LIN {X 0,Y 266.568,Z 546.014,A -85,B 0,C 180,E1 -18838.226,E2 -18838.226} C_VEL
LIN {X 0,Y 268.431,Z 533.162,A -85,B 0,C 180,E1 -18839.08,E2 -18839.08} C_VEL
LIN {X 0,Y 269.683,Z 519.419,A -85,B 0,C 180,E1 -18839.681,E2 -18839.681} C_VEL
LIN {X 0,Y 272.28,Z 465.583,A -85,B 0,C 180,E1 -18841.276,E2 -18841.276} C_VEL
LIN {X 0,Y 269.856,Z 447.877,A -85,B 0,C 180,E1 -18842.351,E2 -18842.351} C_VEL
LIN {X 0,Y 266.008,Z 438.603,A -85,B 0,C 180,E1 -18843.407,E2 -18843.407} C_VEL
LIN {X 0,Y 260.297,Z 427.047,A -85,B 0,C 180,E1 -18844.98,E2 -18844.98} C_VEL
LIN {X 0,Y 255.085,Z 417.615,A -85,B 0,C 180,E1 -18846.5,E2 -18846.5} C_VEL
LIN {X 0,Y 252.805,Z 413.559,A -85,B 0,C 180,E1 -18847.202,E2 -18847.202} C_VEL
LIN {X 0,Y 252.646,Z 413.143,A -85,B 0,C 180,E1 -18847.286,E2 -18847.286} C_VEL
LIN {X 0,Y 250.833,Z 406.63,A -85,B 0,C 180,E1 -18850.843,E2 -18850.843} C_VEL
LIN {X 0,Y 249.024,Z 400.464,A -85,B 0,C 180,E1 -18854.742,E2 -18854.742} C_VEL
LIN {X 0,Y 249.022,Z 400.462,A -85,B 0,C 180,E1 -18857.364,E2 -18857.364} C_VEL
LIN {X 0,Y 249.05,Z 400.458,A -85,B 0,C 180,E1 -18862.201,E2 -18862.201} C_VEL
LIN {X 0,Y 249.05,Z 400.455,A -85,B 0,C 180,E1 -18865.64,E2 -18865.64} C_VEL
LIN {X 0,Y 249.058,Z 400.45,A -85,B 0,C 180,E1 -18869.474,E2 -18869.474} C_VEL
LIN {X 0,Y 249.08,Z 400.447,A -85,B 0,C 180,E1 -18873.163,E2 -18873.163} C_VEL
LIN {X 0,Y 249.086,Z 400.448,A -85,B 0,C 180,E1 -18876.733,E2 -18876.733} C_VEL
LIN {X 0,Y 249.118,Z 400.448,A -85,B 0,C 180,E1 -18880.212,E2 -18880.212} C_VEL
LIN {X 0,Y 249.25,Z 400.438,A -85,B 0,C 180,E1 -18883.622,E2 -18883.622} C_VEL
LIN {X 0,Y 249.26,Z 400.428,A -85,B 0,C 180,E1 -18888.617,E2 -18888.617} C_VEL
LIN {X 0,Y 249.489,Z 400.407,A -85,B 0,C 180,E1 -18891.903,E2 -18891.903} C_VEL
LIN {X 0,Y 249.442,Z 400.404,A -85,B 0,C 180,E1 -18896.77,E2 -18896.77} C_VEL
LIN {X 0,Y 249.729,Z 400.371,A -85,B 0,C 180,E1 -18900,E2 -18900} C_VEL
LIN {X 0,Y 249.442,Z 400.409,A -85,B 0,C 180,E1 -18903.23,E2 -18903.23} C_VEL
LIN {X 0,Y 249.488,Z 400.411,A -85,B 0,C 180,E1 -18908.097,E2 -18908.097} C_VEL
LIN {X 0,Y 249.273,Z 400.636,A -85,B 0,C 180,E1 -18911.795,E2 -18911.795} C_VEL
LIN {X 0,Y 250.357,Z 404.445,A -85,B 0,C 180,E1 -18914.271,E2 -18914.271} C_VEL
LIN {X 0,Y 252.764,Z 408.423,A -85,B 0,C 180,E1 -18915.03,E2 -18915.03} C_VEL
LIN {X 0,Y 254.28,Z 410.816,A -85,B 0,C 180,E1 -18915.49,E2 -18915.49} C_VEL
LIN {X 0,Y 257.244,Z 415.568,A -85,B 0,C 180,E1 -18916.36,E2 -18916.36} C_VEL
LIN {X 0,Y 261.417,Z 422.697,A -85,B 0,C 180,E1 -18917.54,E2 -18917.54} C_VEL
LIN {X 0,Y 267.546,Z 434.619,A -85,B 0,C 180,E1 -18919.194,E2 -18919.194} C_VEL
LIN {X 0,Y 272.807,Z 446.46,A -85,B 0,C 180,E1 -18920.569,E2 -18920.569} C_VEL
LIN {X 0,Y 273.096,Z 448.123,A -85,B 0,C 180,E1 -18920.679,E2 -18920.679} C_VEL
LIN {X 0,Y 269.843,Z 511.083,A -85,B 0,C 180,E1 -18922.55,E2 -18922.55} C_VEL
LIN {X 0,Y 268.607,Z 523.953,A -85,B 0,C 180,E1 -18923.2,E2 -18923.2} C_VEL
LIN {X 0,Y 266.837,Z 537.029,A -85,B 0,C 180,E1 -18924.169,E2 -18924.169} C_VEL
LIN {X 0,Y 264.669,Z 549.571,A -85,B 0,C 180,E1 -18925.463,E2 -18925.463} C_VEL
LIN {X 0,Y 262.411,Z 560.297,A -85,B 0,C 180,E1 -18926.889,E2 -18926.889} C_VEL
LIN {X 0,Y 260.125,Z 569.604,A -85,B 0,C 180,E1 -18928.424,E2 -18928.424} C_VEL
LIN {X 0,Y 257.424,Z 579.801,A -85,B 0,C 180,E1 -18930.551,E2 -18930.551} C_VEL
LIN {X 0,Y 254.954,Z 588.054,A -85,B 0,C 180,E1 -18932.711,E2 -18932.711} C_VEL
LIN {X 0,Y 252.87,Z 594.734,A -85,B 0,C 180,E1 -18934.897,E2 -18934.897} C_VEL
LIN {X 0,Y 250.791,Z 601.307,A -85,B 0,C 180,E1 -18937.658,E2 -18937.658} C_VEL
LIN {X 0,Y 249.183,Z 606.245,A -85,B 0,C 180,E1 -18940.444,E2 -18940.444} C_VEL
LIN {X 0,Y 248.195,Z 609.318,A -85,B 0,C 180,E1 -18942.812,E2 -18942.812} C_VEL
LIN {X 0,Y 247.402,Z 611.514,A -85,B 0,C 180,E1 -18945.25,E2 -18945.25} C_VEL
LIN {X 0,Y 246.873,Z 612.802,A -85,B 0,C 180,E1 -18947.746,E2 -18947.746} C_VEL
LIN {X 0,Y 246.569,Z 613.141,A -85,B 0,C 180,E1 -18950.317,E2 -18950.317} C_VEL
LIN {X 0,Y 246.519,Z 612.309,A -85,B 0,C 180,E1 -18953.222,E2 -18953.222} C_VEL
LIN {X 0,Y 246.722,Z 610.589,A -85,B 0,C 180,E1 -18955.699,E2 -18955.699} C_VEL
LIN {X 0,Y 247.211,Z 607.414,A -85,B 0,C 180,E1 -18958.526,E2 -18958.526} C_VEL
LIN {X 0,Y 247.879,Z 603.161,A -85,B 0,C 180,E1 -18961.182,E2 -18961.182} C_VEL
LIN {X 0,Y 248.794,Z 597.416,A -85,B 0,C 180,E1 -18963.877,E2 -18963.877} C_VEL
LIN {X 0,Y 250.021,Z 590.494,A -85,B 0,C 180,E1 -18966.385,E2 -18966.385} C_VEL
LIN {X 0,Y 251.436,Z 582.526,A -85,B 0,C 180,E1 -18968.691,E2 -18968.691} C_VEL
LIN {X 0,Y 253.046,Z 573.529,A -85,B 0,C 180,E1 -18970.788,E2 -18970.788} C_VEL
LIN {X 0,Y 254.837,Z 562.944,A -85,B 0,C 180,E1 -18972.746,E2 -18972.746} C_VEL
LIN {X 0,Y 256.635,Z 550.86,A -85,B 0,C 180,E1 -18974.512,E2 -18974.512} C_VEL
LIN {X 0,Y 258.123,Z 539.233,A -85,B 0,C 180,E1 -18975.813,E2 -18975.813} C_VEL
LIN {X 0,Y 259.354,Z 527.106,A -85,B 0,C 180,E1 -18976.846,E2 -18976.846} C_VEL
LIN {X 0,Y 260.376,Z 514.047,A -85,B 0,C 180,E1 -18977.632,E2 -18977.632} C_VEL
LIN {X 0,Y 261.108,Z 498.432,A -85,B 0,C 180,E1 -18978.187,E2 -18978.187} C_VEL
LIN {X 0,Y 263.221,Z 439.107,A -85,B 0,C 180,E1 -18979.921,E2 -18979.921} C_VEL
LIN {X 0,Y 259.774,Z 428.453,A -85,B 0,C 180,E1 -18980.596,E2 -18980.596} C_VEL
LIN {X 0,Y 250.616,Z 404.516,A -85,B 0,C 180,E1 -18982.343,E2 -18982.343} C_VEL
LIN {X 0,Y 249.821,Z 402.222,A -85,B 0,C 180,E1 -18982.522,E2 -18982.522} C_VEL
LIN {X 0,Y 249.445,Z 400.414,A -85,B 0,C 180,E1 -18983.324,E2 -18983.324} C_VEL
LIN {X 0,Y 249.679,Z 400.388,A -85,B 0,C 180,E1 -18988.385,E2 -18988.385} C_VEL
LIN {X 0,Y 249.68,Z 400.385,A -85,B 0,C 180,E1 -18991.611,E2 -18991.611} C_VEL
LIN {X 0,Y 249.464,Z 400.408,A -85,B 0,C 180,E1 -18996.468,E2 -18996.468} C_VEL
LIN {X 0,Y 249.426,Z 400.416,A -85,B 0,C 180,E1 -18999.731,E2 -18999.731} C_VEL
LIN {X 0,Y 249.207,Z 400.443,A -85,B 0,C 180,E1 -19004.701,E2 -19004.701} C_VEL
LIN {X 0,Y 249.139,Z 400.447,A -85,B 0,C 180,E1 -19008.075,E2 -19008.075} C_VEL
LIN {X 0,Y 249.085,Z 400.455,A -85,B 0,C 180,E1 -19011.516,E2 -19011.516} C_VEL
LIN {X 0,Y 249.129,Z 400.451,A -85,B 0,C 180,E1 -19015.48,E2 -19015.48} C_VEL
LIN {X 0,Y 249.071,Z 400.45,A -85,B 0,C 180,E1 -19018.987,E2 -19018.987} C_VEL
LIN {X 0,Y 249.033,Z 400.463,A -85,B 0,C 180,E1 -19022.423,E2 -19022.423} C_VEL
LIN {X 0,Y 249.072,Z 400.458,A -85,B 0,C 180,E1 -19026.335,E2 -19026.335} C_VEL
LIN {X 0,Y 249.1,Z 400.46,A -85,B 0,C 180,E1 -19030.05,E2 -19030.05} C_VEL
LIN {X 0,Y 258.347,Z 429.773,A -85,B 0,C 180,E1 -19031.859,E2 -19031.859} C_VEL
LIN {X 0,Y 259.41,Z 437.816,A -85,B 0,C 180,E1 -19032.236,E2 -19032.236} C_VEL
LIN {X 0,Y 256.365,Z 510.289,A -85,B 0,C 180,E1 -19034.889,E2 -19034.889} C_VEL
LIN {X 0,Y 255.661,Z 522.69,A -85,B 0,C 180,E1 -19035.617,E2 -19035.617} C_VEL
LIN {X 0,Y 254.531,Z 536.31,A -85,B 0,C 180,E1 -19036.755,E2 -19036.755} C_VEL
LIN {X 0,Y 253.393,Z 547.649,A -85,B 0,C 180,E1 -19038,E2 -19038} C_VEL
LIN {X 0,Y 252.138,Z 559.069,A -85,B 0,C 180,E1 -19039.604,E2 -19039.604} C_VEL
LIN {X 0,Y 250.863,Z 569.537,A -85,B 0,C 180,E1 -19041.428,E2 -19041.428} C_VEL
LIN {X 0,Y 249.736,Z 578.18,A -85,B 0,C 180,E1 -19043.272,E2 -19043.272} C_VEL
LIN {X 0,Y 248.787,Z 587.017,A -85,B 0,C 180,E1 -19045.599,E2 -19045.599} C_VEL
LIN {X 0,Y 247.951,Z 594.174,A -85,B 0,C 180,E1 -19047.926,E2 -19047.926} C_VEL
LIN {X 0,Y 247.385,Z 599.773,A -85,B 0,C 180,E1 -19050.187,E2 -19050.187} C_VEL
LIN {X 0,Y 246.982,Z 605.008,A -85,B 0,C 180,E1 -19052.916,E2 -19052.916} C_VEL
LIN {X 0,Y 246.573,Z 608.969,A -85,B 0,C 180,E1 -19055.789,E2 -19055.789} C_VEL
LIN {X 0,Y 246.514,Z 611.155,A -85,B 0,C 180,E1 -19058.151,E2 -19058.151} C_VEL
LIN {X 0,Y 245.924,Z 612.139,A -85,B 0,C 180,E1 -19059.499,E2 -19059.499} C_VEL
LIN {X 0,Y 243.285,Z 613.028,A -85,B 0,C 180,E1 -19061.73,E2 -19061.73} C_VEL
LIN {X 0,Y 241.181,Z 613.124,A -85,B 0,C 180,E1 -19063.556,E2 -19063.556} C_VEL
LIN {X 0,Y 240.493,Z 612.898,A -85,B 0,C 180,E1 -19064.962,E2 -19064.962} C_VEL
LIN {X 0,Y 240.551,Z 612.723,A -85,B 0,C 180,E1 -19065.434,E2 -19065.434} C_VEL
LIN {X 0,Y 241.643,Z 611.334,A -85,B 0,C 180,E1 -19068.253,E2 -19068.253} C_VEL
LIN {X 0,Y 242.589,Z 609.736,A -85,B 0,C 180,E1 -19070.051,E2 -19070.051} C_VEL
LIN {X 0,Y 244.269,Z 606.633,A -85,B 0,C 180,E1 -19072.561,E2 -19072.561} C_VEL
LIN {X 0,Y 246.742,Z 601.642,A -85,B 0,C 180,E1 -19075.463,E2 -19075.463} C_VEL
LIN {X 0,Y 249.43,Z 595.792,A -85,B 0,C 180,E1 -19077.981,E2 -19077.981} C_VEL
LIN {X 0,Y 252.714,Z 588.031,A -85,B 0,C 180,E1 -19080.542,E2 -19080.542} C_VEL
LIN {X 0,Y 256.055,Z 579.512,A -85,B 0,C 180,E1 -19082.753,E2 -19082.753} C_VEL
LIN {X 0,Y 259.357,Z 570.212,A -85,B 0,C 180,E1 -19084.663,E2 -19084.663} C_VEL
LIN {X 0,Y 262.551,Z 560.035,A -85,B 0,C 180,E1 -19086.339,E2 -19086.339} C_VEL
LIN {X 0,Y 265.555,Z 548.889,A -85,B 0,C 180,E1 -19087.795,E2 -19087.795} C_VEL
LIN {X 0,Y 268.599,Z 535.466,A -85,B 0,C 180,E1 -19089.137,E2 -19089.137} C_VEL
LIN {X 0,Y 270.877,Z 522.644,A -85,B 0,C 180,E1 -19090.082,E2 -19090.082} C_VEL
LIN {X 0,Y 272.668,Z 509.13,A -85,B 0,C 180,E1 -19090.776,E2 -19090.776} C_VEL
LIN {X 0,Y 277.82,Z 456.002,A -85,B 0,C 180,E1 -19092.755,E2 -19092.755} C_VEL
LIN {X 0,Y 275.399,Z 449.786,A -85,B 0,C 180,E1 -19093.86,E2 -19093.86} C_VEL
LIN {X 0,Y 271.486,Z 442.226,A -85,B 0,C 180,E1 -19095.629,E2 -19095.629} C_VEL
LIN {X 0,Y 267.363,Z 434.936,A -85,B 0,C 180,E1 -19097.722,E2 -19097.722} C_VEL
LIN {X 0,Y 264.428,Z 430.395,A -85,B 0,C 180,E1 -19099.372,E2 -19099.372} C_VEL
LIN {X 0,Y 261.772,Z 426.449,A -85,B 0,C 180,E1 -19101.099,E2 -19101.099} C_VEL
LIN {X 0,Y 258.771,Z 422.149,A -85,B 0,C 180,E1 -19103.407,E2 -19103.407} C_VEL
LIN {X 0,Y 255.488,Z 417.838,A -85,B 0,C 180,E1 -19106.772,E2 -19106.772} C_VEL
LIN {X 0,Y 253.639,Z 416.042,A -85,B 0,C 180,E1 -19109.631,E2 -19109.631} C_VEL
LIN {X 0,Y 252.844,Z 415.227,A -85,B 0,C 180,E1 -19111.879,E2 -19111.879} C_VEL
LIN {X 0,Y 252.7,Z 415.157,A -85,B 0,C 180,E1 -19115.181,E2 -19115.181} C_VEL
LIN {X 0,Y 253.771,Z 416.505,A -85,B 0,C 180,E1 -19118.544,E2 -19118.544} C_VEL
LIN {X 0,Y 255.625,Z 418.278,A -85,B 0,C 180,E1 -19121.205,E2 -19121.205} C_VEL
LIN {X 0,Y 258.033,Z 421.957,A -85,B 0,C 180,E1 -19123.81,E2 -19123.81} C_VEL
LIN {X 0,Y 259.615,Z 423.892,A -85,B 0,C 180,E1 -19125.133,E2 -19125.133} C_VEL
LIN {X 0,Y 261.946,Z 427.27,A -85,B 0,C 180,E1 -19126.84,E2 -19126.84} C_VEL
LIN {X 0,Y 265.527,Z 432.606,A -85,B 0,C 180,E1 -19129.073,E2 -19129.073} C_VEL
LIN {X 0,Y 268.273,Z 436.986,A -85,B 0,C 180,E1 -19130.574,E2 -19130.574} C_VEL
LIN {X 0,Y 271.957,Z 443.193,A -85,B 0,C 180,E1 -19132.381,E2 -19132.381} C_VEL
LIN {X 0,Y 274.992,Z 452.547,A -85,B 0,C 180,E1 -19134.001,E2 -19134.001} C_VEL
LIN {X 0,Y 275.778,Z 455.958,A -85,B 0,C 180,E1 -19134.463,E2 -19134.463} C_VEL
LIN {X 0,Y 276.461,Z 468.834,A -85,B 0,C 180,E1 -19135.487,E2 -19135.487} C_VEL
LIN {X 0,Y 270.924,Z 524.638,A -85,B 0,C 180,E1 -19137.657,E2 -19137.657} C_VEL
LIN {X 0,Y 268.618,Z 538.606,A -85,B 0,C 180,E1 -19138.451,E2 -19138.451} C_VEL
LIN {X 0,Y 265.527,Z 552.57,A -85,B 0,C 180,E1 -19139.591,E2 -19139.591} C_VEL
LIN {X 0,Y 262.393,Z 564.674,A -85,B 0,C 180,E1 -19140.96,E2 -19140.96} C_VEL
LIN {X 0,Y 258.685,Z 576.776,A -85,B 0,C 180,E1 -19142.715,E2 -19142.715} C_VEL
LIN {X 0,Y 255.013,Z 587.409,A -85,B 0,C 180,E1 -19144.714,E2 -19144.714} C_VEL
LIN {X 0,Y 252.05,Z 595.35,A -85,B 0,C 180,E1 -19146.591,E2 -19146.591} C_VEL
LIN {X 0,Y 249.036,Z 603.053,A -85,B 0,C 180,E1 -19148.852,E2 -19148.852} C_VEL
LIN {X 0,Y 246.865,Z 608.633,A -85,B 0,C 180,E1 -19150.892,E2 -19150.892} C_VEL
LIN {X 0,Y 244.527,Z 613.978,A -85,B 0,C 180,E1 -19153.299,E2 -19153.299} C_VEL
LIN {X 0,Y 242.666,Z 618.147,A -85,B 0,C 180,E1 -19155.751,E2 -19155.751} C_VEL
LIN {X 0,Y 241.36,Z 621.281,A -85,B 0,C 180,E1 -19158.241,E2 -19158.241} C_VEL
LIN {X 0,Y 240.717,Z 622.821,A -85,B 0,C 180,E1 -19159.913,E2 -19159.913} C_VEL
LIN {X 0,Y 239.994,Z 624.652,A -85,B 0,C 180,E1 -19163.275,E2 -19163.275} C_VEL
LIN {X 0,Y 239.838,Z 624.974,A -85,B 0,C 180,E1 -19165.076,E2 -19165.076} C_VEL
LIN {X 0,Y 239.812,Z 624.837,A -85,B 0,C 180,E1 -19166.642,E2 -19166.642} C_VEL
LIN {X 0,Y 239.913,Z 626.397,A -85,B 0,C 180,E1 -19170.002,E2 -19170.002} C_VEL
LIN {X 0,Y 239.831,Z 626.688,A -85,B 0,C 180,E1 -19171.681,E2 -19171.681} C_VEL
LIN {X 0,Y 239.791,Z 626.174,A -85,B 0,C 180,E1 -19174.794,E2 -19174.794} C_VEL
LIN {X 0,Y 239.954,Z 625.13,A -85,B 0,C 180,E1 -19176.73,E2 -19176.73} C_VEL
LIN {X 0,Y 240.672,Z 622.058,A -85,B 0,C 180,E1 -19180.093,E2 -19180.093} C_VEL
LIN {X 0,Y 241.624,Z 618.594,A -85,B 0,C 180,E1 -19182.602,E2 -19182.602} C_VEL
LIN {X 0,Y 242.992,Z 614.064,A -85,B 0,C 180,E1 -19185.09,E2 -19185.09} C_VEL
LIN {X 0,Y 245.297,Z 607.243,A -85,B 0,C 180,E1 -19187.941,E2 -19187.941} C_VEL
LIN {X 0,Y 247.616,Z 599.356,A -85,B 0,C 180,E1 -19190.507,E2 -19190.507} C_VEL
LIN {X 0,Y 250.202,Z 590.762,A -85,B 0,C 180,E1 -19192.722,E2 -19192.722} C_VEL
LIN {X 0,Y 252.924,Z 581.377,A -85,B 0,C 180,E1 -19194.635,E2 -19194.635} C_VEL
LIN {X 0,Y 255.855,Z 569.765,A -85,B 0,C 180,E1 -19196.513,E2 -19196.513} C_VEL
LIN {X 0,Y 258.453,Z 558.012,A -85,B 0,C 180,E1 -19197.976,E2 -19197.976} C_VEL
LIN {X 0,Y 260.77,Z 545.587,A -85,B 0,C 180,E1 -19199.133,E2 -19199.133} C_VEL
LIN {X 0,Y 262.745,Z 532.643,A -85,B 0,C 180,E1 -19199.993,E2 -19199.993} C_VEL
LIN {X 0,Y 264.018,Z 518.7,A -85,B 0,C 180,E1 -19200.606,E2 -19200.606} C_VEL
LIN {X 0,Y 266.594,Z 466.135,A -85,B 0,C 180,E1 -19202.206,E2 -19202.206} C_VEL
LIN {X 0,Y 264.479,Z 450.382,A -85,B 0,C 180,E1 -19203.214,E2 -19203.214} C_VEL
LIN {X 0,Y 259.935,Z 439.758,A -85,B 0,C 180,E1 -19204.521,E2 -19204.521} C_VEL
LIN {X 0,Y 253.807,Z 427.521,A -85,B 0,C 180,E1 -19206.341,E2 -19206.341} C_VEL
LIN {X 0,Y 250.372,Z 421.599,A -85,B 0,C 180,E1 -19207.396,E2 -19207.396} C_VEL
LIN {X 0,Y 247.885,Z 417.319,A -85,B 0,C 180,E1 -19208.199,E2 -19208.199} C_VEL
LIN {X 0,Y 245.301,Z 412.722,A -85,B 0,C 180,E1 -19209.154,E2 -19209.154} C_VEL
LIN {X 0,Y 243.583,Z 406.903,A -85,B 0,C 180,E1 -19212.63,E2 -19212.63} C_VEL
LIN {X 0,Y 241.937,Z 401.348,A -85,B 0,C 180,E1 -19216.369,E2 -19216.369} C_VEL
LIN {X 0,Y 241.962,Z 401.339,A -85,B 0,C 180,E1 -19220.282,E2 -19220.282} C_VEL
LIN {X 0,Y 241.995,Z 401.342,A -85,B 0,C 180,E1 -19224.49,E2 -19224.49} C_VEL
LIN {X 0,Y 241.981,Z 401.338,A -85,B 0,C 180,E1 -19228.481,E2 -19228.481} C_VEL
LIN {X 0,Y 242.015,Z 401.332,A -85,B 0,C 180,E1 -19232.314,E2 -19232.314} C_VEL
LIN {X 0,Y 242.064,Z 401.328,A -85,B 0,C 180,E1 -19236.017,E2 -19236.017} C_VEL
LIN {X 0,Y 242.045,Z 401.336,A -85,B 0,C 180,E1 -19239.609,E2 -19239.609} C_VEL
LIN {X 0,Y 242.171,Z 401.32,A -85,B 0,C 180,E1 -19243.279,E2 -19243.279} C_VEL
LIN {X 0,Y 242.194,Z 401.311,A -85,B 0,C 180,E1 -19248.28,E2 -19248.28} C_VEL
LIN {X 0,Y 242.436,Z 401.288,A -85,B 0,C 180,E1 -19251.666,E2 -19251.666} C_VEL
LIN {X 0,Y 242.268,Z 401.308,A -85,B 0,C 180,E1 -19255.007,E2 -19255.007} C_VEL
LIN {X 0,Y 242.643,Z 401.257,A -85,B 0,C 180,E1 -19258.34,E2 -19258.34} C_VEL
LIN {X 0,Y 242.643,Z 401.257,A -85,B 0,C 180,E1 -19261.66,E2 -19261.66} C_VEL
LIN {X 0,Y 242.437,Z 401.281,A -85,B 0,C 180,E1 -19266.722,E2 -19266.722} C_VEL
LIN {X 0,Y 242.34,Z 401.329,A -85,B 0,C 180,E1 -19270.021,E2 -19270.021} C_VEL
LIN {X 0,Y 243.262,Z 404.963,A -85,B 0,C 180,E1 -19272.453,E2 -19272.453} C_VEL
LIN {X 0,Y 246.064,Z 409.288,A -85,B 0,C 180,E1 -19273.419,E2 -19273.419} C_VEL
LIN {X 0,Y 250.565,Z 416.308,A -85,B 0,C 180,E1 -19274.882,E2 -19274.882} C_VEL
LIN {X 0,Y 255.602,Z 424.606,A -85,B 0,C 180,E1 -19276.401,E2 -19276.401} C_VEL
LIN {X 0,Y 261.988,Z 436.923,A -85,B 0,C 180,E1 -19278.241,E2 -19278.241} C_VEL
LIN {X 0,Y 267.348,Z 449.096,A -85,B 0,C 180,E1 -19279.733,E2 -19279.733} C_VEL
LIN {X 0,Y 266.268,Z 472.036,A -85,B 0,C 180,E1 -19280.445,E2 -19280.445} C_VEL
LIN {X 0,Y 264.106,Z 511.487,A -85,B 0,C 180,E1 -19281.656,E2 -19281.656} C_VEL
LIN {X 0,Y 262.807,Z 524.48,A -85,B 0,C 180,E1 -19282.329,E2 -19282.329} C_VEL
LIN {X 0,Y 260.98,Z 537.375,A -85,B 0,C 180,E1 -19283.305,E2 -19283.305} C_VEL
LIN {X 0,Y 258.833,Z 549.258,A -85,B 0,C 180,E1 -19284.544,E2 -19284.544} C_VEL
LIN {X 0,Y 256.412,Z 560.221,A -85,B 0,C 180,E1 -19286.011,E2 -19286.011} C_VEL
LIN {X 0,Y 253.916,Z 570.012,A -85,B 0,C 180,E1 -19287.657,E2 -19287.657} C_VEL
LIN {X 0,Y 251.461,Z 578.97,A -85,B 0,C 180,E1 -19289.55,E2 -19289.55} C_VEL
LIN {X 0,Y 248.545,Z 588.123,A -85,B 0,C 180,E1 -19291.97,E2 -19291.97} C_VEL
LIN {X 0,Y 246.355,Z 594.734,A -85,B 0,C 180,E1 -19294.173,E2 -19294.173} C_VEL
LIN {X 0,Y 244.518,Z 600.118,A -85,B 0,C 180,E1 -19296.408,E2 -19296.408} C_VEL
LIN {X 0,Y 243.058,Z 604.453,A -85,B 0,C 180,E1 -19298.672,E2 -19298.672} C_VEL
LIN {X 0,Y 241.399,Z 609.18,A -85,B 0,C 180,E1 -19302.038,E2 -19302.038} C_VEL
LIN {X 0,Y 240.507,Z 611.498,A -85,B 0,C 180,E1 -19304.533,E2 -19304.533} C_VEL
LIN {X 0,Y 239.816,Z 613.053,A -85,B 0,C 180,E1 -19307.618,E2 -19307.618} C_VEL
LIN {X 0,Y 239.507,Z 613.374,A -85,B 0,C 180,E1 -19309.79,E2 -19309.79} C_VEL
LIN {X 0,Y 239.401,Z 612.831,A -85,B 0,C 180,E1 -19312.433,E2 -19312.433} C_VEL
LIN {X 0,Y 239.572,Z 611.171,A -85,B 0,C 180,E1 -19315.226,E2 -19315.226} C_VEL
LIN {X 0,Y 240.037,Z 608.096,A -85,B 0,C 180,E1 -19318.193,E2 -19318.193} C_VEL
LIN {X 0,Y 240.751,Z 603.639,A -85,B 0,C 180,E1 -19321.136,E2 -19321.136} C_VEL
LIN {X 0,Y 241.6,Z 598.536,A -85,B 0,C 180,E1 -19323.663,E2 -19323.663} C_VEL
LIN {X 0,Y 242.722,Z 592.355,A -85,B 0,C 180,E1 -19326.084,E2 -19326.084} C_VEL
LIN {X 0,Y 244.122,Z 584.751,A -85,B 0,C 180,E1 -19328.464,E2 -19328.464} C_VEL
LIN {X 0,Y 245.781,Z 575.944,A -85,B 0,C 180,E1 -19330.67,E2 -19330.67} C_VEL
LIN {X 0,Y 247.518,Z 566.141,A -85,B 0,C 180,E1 -19332.652,E2 -19332.652} C_VEL
LIN {X 0,Y 249.188,Z 555.878,A -85,B 0,C 180,E1 -19334.32,E2 -19334.32} C_VEL
LIN {X 0,Y 250.807,Z 544.253,A -85,B 0,C 180,E1 -19335.805,E2 -19335.805} C_VEL
LIN {X 0,Y 252.27,Z 531.643,A -85,B 0,C 180,E1 -19337.037,E2 -19337.037} C_VEL
LIN {X 0,Y 253.431,Z 518.677,A -85,B 0,C 180,E1 -19337.943,E2 -19337.943} C_VEL
LIN {X 0,Y 254.242,Z 505.414,A -85,B 0,C 180,E1 -19338.538,E2 -19338.538} C_VEL
LIN {X 0,Y 256.641,Z 440.017,A -85,B 0,C 180,E1 -19340.51,E2 -19340.51} C_VEL
LIN {X 0,Y 248.497,Z 417.323,A -85,B 0,C 180,E1 -19342.116,E2 -19342.116} C_VEL
LIN {X 0,Y 242.596,Z 402.349,A -85,B 0,C 180,E1 -19343.344,E2 -19343.344} C_VEL
LIN {X 0,Y 242.359,Z 401.297,A -85,B 0,C 180,E1 -19343.859,E2 -19343.859} C_VEL
LIN {X 0,Y 242.639,Z 401.265,A -85,B 0,C 180,E1 -19348.338,E2 -19348.338} C_VEL
LIN {X 0,Y 242.64,Z 401.262,A -85,B 0,C 180,E1 -19351.658,E2 -19351.658} C_VEL
LIN {X 0,Y 242.437,Z 401.282,A -85,B 0,C 180,E1 -19356.657,E2 -19356.657} C_VEL
LIN {X 0,Y 242.347,Z 401.3,A -85,B 0,C 180,E1 -19360.018,E2 -19360.018} C_VEL
LIN {X 0,Y 242.168,Z 401.319,A -85,B 0,C 180,E1 -19365.138,E2 -19365.138} C_VEL
LIN {X 0,Y 242.072,Z 401.323,A -85,B 0,C 180,E1 -19368.622,E2 -19368.622} C_VEL
LIN {X 0,Y 242.011,Z 401.34,A -85,B 0,C 180,E1 -19372.178,E2 -19372.178} C_VEL
LIN {X 0,Y 242.065,Z 401.326,A -85,B 0,C 180,E1 -19375.836,E2 -19375.836} C_VEL
LIN {X 0,Y 242.005,Z 401.333,A -85,B 0,C 180,E1 -19379.581,E2 -19379.581} C_VEL
LIN {X 0,Y 241.988,Z 401.343,A -85,B 0,C 180,E1 -19383.488,E2 -19383.488} C_VEL
LIN {X 0,Y 242.01,Z 401.341,A -85,B 0,C 180,E1 -19387.575,E2 -19387.575} C_VEL
LIN {X 0,Y 242.044,Z 401.339,A -85,B 0,C 180,E1 -19389.545,E2 -19389.545} C_VEL
LIN {X 0,Y 249.887,Z 425.715,A -85,B 0,C 180,E1 -19391.133,E2 -19391.133} C_VEL
LIN {X 0,Y 251.825,Z 432.71,A -85,B 0,C 180,E1 -19391.546,E2 -19391.546} C_VEL
LIN {X 0,Y 252.582,Z 438.328,A -85,B 0,C 180,E1 -19391.818,E2 -19391.818} C_VEL
LIN {X 0,Y 249.442,Z 510.774,A -85,B 0,C 180,E1 -19394.56,E2 -19394.56} C_VEL
LIN {X 0,Y 248.664,Z 523.331,A -85,B 0,C 180,E1 -19395.328,E2 -19395.328} C_VEL
LIN {X 0,Y 247.528,Z 536.734,A -85,B 0,C 180,E1 -19396.486,E2 -19396.486} C_VEL
LIN {X 0,Y 246.27,Z 548.996,A -85,B 0,C 180,E1 -19397.897,E2 -19397.897} C_VEL
LIN {X 0,Y 245.003,Z 560.145,A -85,B 0,C 180,E1 -19399.533,E2 -19399.533} C_VEL
LIN {X 0,Y 243.749,Z 570.254,A -85,B 0,C 180,E1 -19401.369,E2 -19401.369} C_VEL
LIN {X 0,Y 242.489,Z 579.841,A -85,B 0,C 180,E1 -19403.537,E2 -19403.537} C_VEL
LIN {X 0,Y 241.527,Z 588.431,A -85,B 0,C 180,E1 -19405.934,E2 -19405.934} C_VEL
LIN {X 0,Y 240.719,Z 595.238,A -85,B 0,C 180,E1 -19408.296,E2 -19408.296} C_VEL
LIN {X 0,Y 240.208,Z 601.145,A -85,B 0,C 180,E1 -19410.875,E2 -19410.875} C_VEL
LIN {X 0,Y 239.713,Z 606.438,A -85,B 0,C 180,E1 -19413.91,E2 -19413.91} C_VEL
LIN {X 0,Y 239.504,Z 608.808,A -85,B 0,C 180,E1 -19415.744,E2 -19415.744} C_VEL
LIN {X 0,Y 239.398,Z 611.078,A -85,B 0,C 180,E1 -19418.16,E2 -19418.16} C_VEL
LIN {X 0,Y 239.51,Z 612.221,A -85,B 0,C 180,E1 -19419.874,E2 -19419.874} C_VEL
LIN {X 0,Y 239.946,Z 613.112,A -85,B 0,C 180,E1 -19422.968,E2 -19422.968} C_VEL
LIN {X 0,Y 240.551,Z 612.723,A -85,B 0,C 180,E1 -19425.434,E2 -19425.434} C_VEL
LIN {X 0,Y 240.37,Z 612.261,A -85,B 0,C 180,E1 -19426.836,E2 -19426.836} C_VEL
LIN {X 0,Y 238.52,Z 611.009,A -85,B 0,C 180,E1 -19429.152,E2 -19429.152} C_VEL
LIN {X 0,Y 237.004,Z 609.191,A -85,B 0,C 180,E1 -19431.472,E2 -19431.472} C_VEL
LIN {X 0,Y 237.339,Z 607.608,A -85,B 0,C 180,E1 -19432.846,E2 -19432.846} C_VEL
LIN {X 0,Y 239.666,Z 603.432,A -85,B 0,C 180,E1 -19435.541,E2 -19435.541} C_VEL
LIN {X 0,Y 242.621,Z 597.494,A -85,B 0,C 180,E1 -19438.34,E2 -19438.34} C_VEL
LIN {X 0,Y 246,Z 590.388,A -85,B 0,C 180,E1 -19440.911,E2 -19440.911} C_VEL
LIN {X 0,Y 249.504,Z 582.136,A -85,B 0,C 180,E1 -19443.229,E2 -19443.229} C_VEL
LIN {X 0,Y 253.385,Z 572.109,A -85,B 0,C 180,E1 -19445.431,E2 -19445.431} C_VEL
LIN {X 0,Y 257.008,Z 561.408,A -85,B 0,C 180,E1 -19447.266,E2 -19447.266} C_VEL
LIN {X 0,Y 260.176,Z 550.665,A -85,B 0,C 180,E1 -19448.74,E2 -19448.74} C_VEL
LIN {X 0,Y 263.144,Z 538.765,A -85,B 0,C 180,E1 -19449.998,E2 -19449.998} C_VEL
LIN {X 0,Y 265.826,Z 525.23,A -85,B 0,C 180,E1 -19451.077,E2 -19451.077} C_VEL
LIN {X 0,Y 267.802,Z 511.666,A -85,B 0,C 180,E1 -19451.819,E2 -19451.819} C_VEL
LIN {X 0,Y 273.357,Z 458.874,A -85,B 0,C 180,E1 -19453.832,E2 -19453.832} C_VEL
LIN {X 0,Y 270.772,Z 452.622,A -85,B 0,C 180,E1 -19455.072,E2 -19455.072} C_VEL
LIN {X 0,Y 266.891,Z 445.109,A -85,B 0,C 180,E1 -19457.019,E2 -19457.019} C_VEL
LIN {X 0,Y 263.865,Z 439.602,A -85,B 0,C 180,E1 -19458.744,E2 -19458.744} C_VEL
LIN {X 0,Y 261.787,Z 436.366,A -85,B 0,C 180,E1 -19460.02,E2 -19460.02} C_VEL
LIN {X 0,Y 259.543,Z 432.863,A -85,B 0,C 180,E1 -19461.555,E2 -19461.555} C_VEL
LIN {X 0,Y 256.667,Z 428.644,A -85,B 0,C 180,E1 -19463.901,E2 -19463.901} C_VEL
LIN {X 0,Y 253.731,Z 424.52,A -85,B 0,C 180,E1 -19467.195,E2 -19467.195} C_VEL
LIN {X 0,Y 251.982,Z 422.789,A -85,B 0,C 180,E1 -19470.166,E2 -19470.166} C_VEL
LIN {X 0,Y 251.252,Z 422.055,A -85,B 0,C 180,E1 -19472.953,E2 -19472.953} C_VEL
LIN {X 0,Y 251.404,Z 422.303,A -85,B 0,C 180,E1 -19475.948,E2 -19475.948} C_VEL
LIN {X 0,Y 253.539,Z 424.567,A -85,B 0,C 180,E1 -19480.376,E2 -19480.376} C_VEL
LIN {X 0,Y 254.089,Z 425.443,A -85,B 0,C 180,E1 -19481.147,E2 -19481.147} C_VEL
LIN {X 0,Y 256.599,Z 429.109,A -85,B 0,C 180,E1 -19483.852,E2 -19483.852} C_VEL
LIN {X 0,Y 257.638,Z 430.512,A -85,B 0,C 180,E1 -19484.752,E2 -19484.752} C_VEL
LIN {X 0,Y 260.994,Z 435.664,A -85,B 0,C 180,E1 -19487.281,E2 -19487.281} C_VEL
LIN {X 0,Y 263.165,Z 439.105,A -85,B 0,C 180,E1 -19488.662,E2 -19488.662} C_VEL
LIN {X 0,Y 265.862,Z 443.65,A -85,B 0,C 180,E1 -19490.227,E2 -19490.227} C_VEL
LIN {X 0,Y 268.745,Z 448.915,A -85,B 0,C 180,E1 -19491.73,E2 -19491.73} C_VEL
LIN {X 0,Y 271.591,Z 458.563,A -85,B 0,C 180,E1 -19493.394,E2 -19493.394} C_VEL
LIN {X 0,Y 272.014,Z 470.266,A -85,B 0,C 180,E1 -19494.36,E2 -19494.36} C_VEL
LIN {X 0,Y 266.398,Z 523.966,A -85,B 0,C 180,E1 -19496.473,E2 -19496.473} C_VEL
LIN {X 0,Y 264.004,Z 537.881,A -85,B 0,C 180,E1 -19497.269,E2 -19497.269} C_VEL
LIN {X 0,Y 260.976,Z 550.939,A -85,B 0,C 180,E1 -19498.326,E2 -19498.326} C_VEL
LIN {X 0,Y 257.631,Z 563.395,A -85,B 0,C 180,E1 -19499.693,E2 -19499.693} C_VEL
LIN {X 0,Y 253.677,Z 575.657,A -85,B 0,C 180,E1 -19501.454,E2 -19501.454} C_VEL
LIN {X 0,Y 250.105,Z 585.524,A -85,B 0,C 180,E1 -19503.284,E2 -19503.284} C_VEL
LIN {X 0,Y 246.251,Z 595.175,A -85,B 0,C 180,E1 -19505.557,E2 -19505.557} C_VEL
LIN {X 0,Y 242.914,Z 603.046,A -85,B 0,C 180,E1 -19507.909,E2 -19507.909} C_VEL
LIN {X 0,Y 240.216,Z 609.367,A -85,B 0,C 180,E1 -19510.341,E2 -19510.341} C_VEL
LIN {X 0,Y 237.769,Z 614.48,A -85,B 0,C 180,E1 -19512.81,E2 -19512.81} C_VEL
LIN {X 0,Y 235.773,Z 618.484,A -85,B 0,C 180,E1 -19515.325,E2 -19515.325} C_VEL
LIN {X 0,Y 234.393,Z 621.451,A -85,B 0,C 180,E1 -19517.887,E2 -19517.887} C_VEL
LIN {X 0,Y 233.219,Z 623.918,A -85,B 0,C 180,E1 -19521.336,E2 -19521.336} C_VEL
LIN {X 0,Y 232.921,Z 624.555,A -85,B 0,C 180,E1 -19523.07,E2 -19523.07} C_VEL
LIN {X 0,Y 232.731,Z 624.722,A -85,B 0,C 180,E1 -19525.228,E2 -19525.228} C_VEL
LIN {X 0,Y 232.731,Z 624.569,A -85,B 0,C 180,E1 -19526.973,E2 -19526.973} C_VEL
LIN {X 0,Y 232.822,Z 626.146,A -85,B 0,C 180,E1 -19530.002,E2 -19530.002} C_VEL
LIN {X 0,Y 232.742,Z 626.469,A -85,B 0,C 180,E1 -19531.733,E2 -19531.733} C_VEL
LIN {X 0,Y 232.732,Z 625.938,A -85,B 0,C 180,E1 -19535.2,E2 -19535.2} C_VEL
LIN {X 0,Y 232.892,Z 625.043,A -85,B 0,C 180,E1 -19536.935,E2 -19536.935} C_VEL
LIN {X 0,Y 233.67,Z 622.038,A -85,B 0,C 180,E1 -19540.399,E2 -19540.399} C_VEL
LIN {X 0,Y 234.66,Z 618.643,A -85,B 0,C 180,E1 -19542.983,E2 -19542.983} C_VEL
LIN {X 0,Y 236.151,Z 614.186,A -85,B 0,C 180,E1 -19545.538,E2 -19545.538} C_VEL
LIN {X 0,Y 238.553,Z 607.516,A -85,B 0,C 180,E1 -19548.466,E2 -19548.466} C_VEL
LIN {X 0,Y 240.901,Z 600.076,A -85,B 0,C 180,E1 -19551.003,E2 -19551.003} C_VEL
LIN {X 0,Y 243.695,Z 591.296,A -85,B 0,C 180,E1 -19553.364,E2 -19553.364} C_VEL
LIN {X 0,Y 246.54,Z 582.116,A -85,B 0,C 180,E1 -19555.317,E2 -19555.317} C_VEL
LIN {X 0,Y 249.578,Z 570.707,A -85,B 0,C 180,E1 -19557.234,E2 -19557.234} C_VEL
LIN {X 0,Y 252.275,Z 559.283,A -85,B 0,C 180,E1 -19558.724,E2 -19558.724} C_VEL
LIN {X 0,Y 254.848,Z 546.283,A -85,B 0,C 180,E1 -19559.991,E2 -19559.991} C_VEL
LIN {X 0,Y 256.875,Z 533.72,A -85,B 0,C 180,E1 -19560.865,E2 -19560.865} C_VEL
LIN {X 0,Y 258.292,Z 520.295,A -85,B 0,C 180,E1 -19561.502,E2 -19561.502} C_VEL
LIN {X 0,Y 261.135,Z 467.707,A -85,B 0,C 180,E1 -19563.133,E2 -19563.133} C_VEL
LIN {X 0,Y 259.301,Z 453.36,A -85,B 0,C 180,E1 -19564.075,E2 -19564.075} C_VEL
LIN {X 0,Y 255.078,Z 443.476,A -85,B 0,C 180,E1 -19565.354,E2 -19565.354} C_VEL
LIN {X 0,Y 249.295,Z 431.757,A -85,B 0,C 180,E1 -19567.175,E2 -19567.175} C_VEL
LIN {X 0,Y 244.323,Z 422.817,A -85,B 0,C 180,E1 -19568.837,E2 -19568.837} C_VEL
LIN {X 0,Y 241.013,Z 417.544,A -85,B 0,C 180,E1 -19569.992,E2 -19569.992} C_VEL
LIN {X 0,Y 238.266,Z 413.211,A -85,B 0,C 180,E1 -19571.007,E2 -19571.007} C_VEL
LIN {X 0,Y 237.888,Z 412.305,A -85,B 0,C 180,E1 -19571.278,E2 -19571.278} C_VEL
LIN {X 0,Y 236.489,Z 407.369,A -85,B 0,C 180,E1 -19574.501,E2 -19574.501} C_VEL
LIN {X 0,Y 234.889,Z 402.228,A -85,B 0,C 180,E1 -19578.421,E2 -19578.421} C_VEL
LIN {X 0,Y 234.925,Z 402.221,A -85,B 0,C 180,E1 -19581.08,E2 -19581.08} C_VEL
LIN {X 0,Y 234.937,Z 402.214,A -85,B 0,C 180,E1 -19585.363,E2 -19585.363} C_VEL
LIN {X 0,Y 234.938,Z 402.209,A -85,B 0,C 180,E1 -19589.433,E2 -19589.433} C_VEL
LIN {X 0,Y 235.001,Z 402.201,A -85,B 0,C 180,E1 -19593.795,E2 -19593.795} C_VEL
LIN {X 0,Y 235.019,Z 402.209,A -85,B 0,C 180,E1 -19598.971,E2 -19598.971} C_VEL
LIN {X 0,Y 235.104,Z 402.199,A -85,B 0,C 180,E1 -19603.06,E2 -19603.06} C_VEL
LIN {X 0,Y 235.154,Z 402.191,A -85,B 0,C 180,E1 -19607.924,E2 -19607.924} C_VEL
LIN {X 0,Y 235.385,Z 402.165,A -85,B 0,C 180,E1 -19611.414,E2 -19611.414} C_VEL
LIN {X 0,Y 235.412,Z 402.15,A -85,B 0,C 180,E1 -19613.142,E2 -19613.142} C_VEL
LIN {X 0,Y 235.603,Z 402.133,A -85,B 0,C 180,E1 -19618.291,E2 -19618.291} C_VEL
LIN {X 0,Y 235.603,Z 402.134,A -85,B 0,C 180,E1 -19621.71,E2 -19621.71} C_VEL
LIN {X 0,Y 235.384,Z 402.166,A -85,B 0,C 180,E1 -19627.938,E2 -19627.938} C_VEL
LIN {X 0,Y 236.155,Z 405.311,A -85,B 0,C 180,E1 -19630.394,E2 -19630.394} C_VEL
LIN {X 0,Y 238.23,Z 408.723,A -85,B 0,C 180,E1 -19631.217,E2 -19631.217} C_VEL
LIN {X 0,Y 240.051,Z 411.067,A -85,B 0,C 180,E1 -19631.88,E2 -19631.88} C_VEL
LIN {X 0,Y 246.088,Z 420.27,A -85,B 0,C 180,E1 -19633.97,E2 -19633.97} C_VEL
LIN {X 0,Y 252.467,Z 431.309,A -85,B 0,C 180,E1 -19636.008,E2 -19636.008} C_VEL
LIN {X 0,Y 258.155,Z 442.889,A -85,B 0,C 180,E1 -19637.739,E2 -19637.739} C_VEL
LIN {X 0,Y 261.952,Z 451.736,A -85,B 0,C 180,E1 -19638.844,E2 -19638.844} C_VEL
LIN {X 0,Y 258.526,Z 511.52,A -85,B 0,C 180,E1 -19640.696,E2 -19640.696} C_VEL
LIN {X 0,Y 257.175,Z 524.358,A -85,B 0,C 180,E1 -19641.367,E2 -19641.367} C_VEL
LIN {X 0,Y 255.276,Z 537.214,A -85,B 0,C 180,E1 -19642.347,E2 -19642.347} C_VEL
LIN {X 0,Y 253.066,Z 548.954,A -85,B 0,C 180,E1 -19643.583,E2 -19643.583} C_VEL
LIN {X 0,Y 250.541,Z 559.903,A -85,B 0,C 180,E1 -19645.056,E2 -19645.056} C_VEL
LIN {X 0,Y 247.834,Z 570.187,A -85,B 0,C 180,E1 -19646.809,E2 -19646.809} C_VEL
LIN {X 0,Y 245.35,Z 578.678,A -85,B 0,C 180,E1 -19648.616,E2 -19648.616} C_VEL
LIN {X 0,Y 242.544,Z 587.171,A -85,B 0,C 180,E1 -19650.859,E2 -19650.859} C_VEL
LIN {X 0,Y 240.092,Z 594.064,A -85,B 0,C 180,E1 -19653.134,E2 -19653.134} C_VEL
LIN {X 0,Y 238.072,Z 599.712,A -85,B 0,C 180,E1 -19655.475,E2 -19655.475} C_VEL
LIN {X 0,Y 236.445,Z 604.262,A -85,B 0,C 180,E1 -19657.857,E2 -19657.857} C_VEL
LIN {X 0,Y 235.098,Z 607.838,A -85,B 0,C 180,E1 -19660.254,E2 -19660.254} C_VEL
LIN {X 0,Y 234.04,Z 610.481,A -85,B 0,C 180,E1 -19662.63,E2 -19662.63} C_VEL
LIN {X 0,Y 233.001,Z 612.811,A -85,B 0,C 180,E1 -19666.07,E2 -19666.07} C_VEL
LIN {X 0,Y 232.472,Z 613.554,A -85,B 0,C 180,E1 -19669.095,E2 -19669.095} C_VEL
LIN {X 0,Y 232.301,Z 613.158,A -85,B 0,C 180,E1 -19671.869,E2 -19671.869} C_VEL
LIN {X 0,Y 232.436,Z 611.528,A -85,B 0,C 180,E1 -19674.934,E2 -19674.934} C_VEL
LIN {X 0,Y 232.825,Z 608.924,A -85,B 0,C 180,E1 -19677.694,E2 -19677.694} C_VEL
LIN {X 0,Y 233.38,Z 605.784,A -85,B 0,C 180,E1 -19680.041,E2 -19680.041} C_VEL
LIN {X 0,Y 234.353,Z 599.98,A -85,B 0,C 180,E1 -19683.265,E2 -19683.265} C_VEL
LIN {X 0,Y 235.695,Z 592.751,A -85,B 0,C 180,E1 -19686.26,E2 -19686.26} C_VEL
LIN {X 0,Y 237.122,Z 585.214,A -85,B 0,C 180,E1 -19688.709,E2 -19688.709} C_VEL
LIN {X 0,Y 238.944,Z 575.839,A -85,B 0,C 180,E1 -19691.121,E2 -19691.121} C_VEL
LIN {X 0,Y 240.869,Z 565.406,A -85,B 0,C 180,E1 -19693.262,E2 -19693.262} C_VEL
LIN {X 0,Y 242.715,Z 553.922,A -85,B 0,C 180,E1 -19695.107,E2 -19695.107} C_VEL
LIN {X 0,Y 244.425,Z 542.051,A -85,B 0,C 180,E1 -19696.594,E2 -19696.594} C_VEL
LIN {X 0,Y 245.815,Z 529.628,A -85,B 0,C 180,E1 -19697.769,E2 -19697.769} C_VEL
LIN {X 0,Y 246.994,Z 516.182,A -85,B 0,C 180,E1 -19698.665,E2 -19698.665} C_VEL
LIN {X 0,Y 247.746,Z 502.926,A -85,B 0,C 180,E1 -19699.217,E2 -19699.217} C_VEL
LIN {X 0,Y 250.092,Z 441.448,A -85,B 0,C 180,E1 -19701.112,E2 -19701.112} C_VEL
LIN {X 0,Y 240.933,Z 416.334,A -85,B 0,C 180,E1 -19702.966,E2 -19702.966} C_VEL
LIN {X 0,Y 235.968,Z 404.432,A -85,B 0,C 180,E1 -19703.98,E2 -19703.98} C_VEL
LIN {X 0,Y 235.346,Z 402.6,A -85,B 0,C 180,E1 -19704.16,E2 -19704.16} C_VEL
LIN {X 0,Y 235.246,Z 402.181,A -85,B 0,C 180,E1 -19704.426,E2 -19704.426} C_VEL
LIN {X 0,Y 235.598,Z 402.142,A -85,B 0,C 180,E1 -19708.288,E2 -19708.288} C_VEL
LIN {X 0,Y 235.6,Z 402.14,A -85,B 0,C 180,E1 -19711.707,E2 -19711.707} C_VEL
LIN {X 0,Y 235.408,Z 402.157,A -85,B 0,C 180,E1 -19716.856,E2 -19716.856} C_VEL
LIN {X 0,Y 235.255,Z 402.182,A -85,B 0,C 180,E1 -19720.323,E2 -19720.323} C_VEL
LIN {X 0,Y 235.114,Z 402.199,A -85,B 0,C 180,E1 -19725.604,E2 -19725.604} C_VEL
LIN {X 0,Y 235.008,Z 402.203,A -85,B 0,C 180,E1 -19729.203,E2 -19729.203} C_VEL
LIN {X 0,Y 234.959,Z 402.216,A -85,B 0,C 180,E1 -19732.88,E2 -19732.88} C_VEL
LIN {X 0,Y 234.966,Z 402.206,A -85,B 0,C 180,E1 -19736.655,E2 -19736.655} C_VEL
LIN {X 0,Y 234.92,Z 402.218,A -85,B 0,C 180,E1 -19740.566,E2 -19740.566} C_VEL
LIN {X 0,Y 234.957,Z 402.216,A -85,B 0,C 180,E1 -19744.63,E2 -19744.63} C_VEL
LIN {X 0,Y 234.999,Z 402.212,A -85,B 0,C 180,E1 -19749.026,E2 -19749.026} C_VEL
LIN {X 0,Y 240.929,Z 420.062,A -85,B 0,C 180,E1 -19750.261,E2 -19750.261} C_VEL
LIN {X 0,Y 245.072,Z 433.85,A -85,B 0,C 180,E1 -19751.128,E2 -19751.128} C_VEL
LIN {X 0,Y 245.736,Z 439.338,A -85,B 0,C 180,E1 -19751.401,E2 -19751.401} C_VEL
LIN {X 0,Y 242.539,Z 510.325,A -85,B 0,C 180,E1 -19754.178,E2 -19754.178} C_VEL
LIN {X 0,Y 241.697,Z 523.629,A -85,B 0,C 180,E1 -19755.012,E2 -19755.012} C_VEL
LIN {X 0,Y 240.52,Z 537.185,A -85,B 0,C 180,E1 -19756.227,E2 -19756.227} C_VEL
LIN {X 0,Y 239.349,Z 548.187,A -85,B 0,C 180,E1 -19757.518,E2 -19757.518} C_VEL
LIN {X 0,Y 238.049,Z 559.561,A -85,B 0,C 180,E1 -19759.216,E2 -19759.216} C_VEL
LIN {X 0,Y 236.782,Z 569.444,A -85,B 0,C 180,E1 -19761.036,E2 -19761.036} C_VEL
LIN {X 0,Y 235.674,Z 577.592,A -85,B 0,C 180,E1 -19762.852,E2 -19762.852} C_VEL
LIN {X 0,Y 234.648,Z 586.623,A -85,B 0,C 180,E1 -19765.314,E2 -19765.314} C_VEL
LIN {X 0,Y 233.797,Z 593.828,A -85,B 0,C 180,E1 -19767.753,E2 -19767.753} C_VEL
LIN {X 0,Y 233.22,Z 599.585,A -85,B 0,C 180,E1 -19770.162,E2 -19770.162} C_VEL
LIN {X 0,Y 232.774,Z 605.025,A -85,B 0,C 180,E1 -19773.071,E2 -19773.071} C_VEL
LIN {X 0,Y 232.457,Z 607.889,A -85,B 0,C 180,E1 -19775.089,E2 -19775.089} C_VEL
LIN {X 0,Y 232.322,Z 609.887,A -85,B 0,C 180,E1 -19776.842,E2 -19776.842} C_VEL
LIN {X 0,Y 232.404,Z 612.077,A -85,B 0,C 180,E1 -19779.62,E2 -19779.62} C_VEL
LIN {X 0,Y 232.756,Z 613.182,A -85,B 0,C 180,E1 -19782.425,E2 -19782.425} C_VEL
LIN {X 0,Y 233.493,Z 613.1,A -85,B 0,C 180,E1 -19785.576,E2 -19785.576} C_VEL
LIN {X 0,Y 234.368,Z 612.218,A -85,B 0,C 180,E1 -19787.883,E2 -19787.883} C_VEL
LIN {X 0,Y 235.461,Z 610.682,A -85,B 0,C 180,E1 -19790.04,E2 -19790.04} C_VEL
LIN {X 0,Y 237.339,Z 607.608,A -85,B 0,C 180,E1 -19792.846,E2 -19792.846} C_VEL
LIN {X 0,Y 237.785,Z 605.853,A -85,B 0,C 180,E1 -19794.204,E2 -19794.204} C_VEL
LIN {X 0,Y 236.966,Z 602.77,A -85,B 0,C 180,E1 -19796.474,E2 -19796.474} C_VEL
LIN {X 0,Y 236.474,Z 599.074,A -85,B 0,C 180,E1 -19798.692,E2 -19798.692} C_VEL
LIN {X 0,Y 237.398,Z 596.343,A -85,B 0,C 180,E1 -19799.935,E2 -19799.935} C_VEL
LIN {X 0,Y 241.012,Z 588.938,A -85,B 0,C 180,E1 -19802.507,E2 -19802.507} C_VEL
LIN {X 0,Y 245.082,Z 579.928,A -85,B 0,C 180,E1 -19804.935,E2 -19804.935} C_VEL
LIN {X 0,Y 249.172,Z 569.651,A -85,B 0,C 180,E1 -19807.088,E2 -19807.088} C_VEL
LIN {X 0,Y 252.8,Z 559.289,A -85,B 0,C 180,E1 -19808.795,E2 -19808.795} C_VEL
LIN {X 0,Y 256.402,Z 547.151,A -85,B 0,C 180,E1 -19810.343,E2 -19810.343} C_VEL
LIN {X 0,Y 259.426,Z 534.964,A -85,B 0,C 180,E1 -19811.543,E2 -19811.543} C_VEL
LIN {X 0,Y 261.608,Z 523.938,A -85,B 0,C 180,E1 -19812.37,E2 -19812.37} C_VEL
LIN {X 0,Y 263.546,Z 511.246,A -85,B 0,C 180,E1 -19813.052,E2 -19813.052} C_VEL
LIN {X 0,Y 268.992,Z 461.617,A -85,B 0,C 180,E1 -19814.978,E2 -19814.978} C_VEL
LIN {X 0,Y 265.902,Z 454.616,A -85,B 0,C 180,E1 -19816.6,E2 -19816.6} C_VEL
LIN {X 0,Y 261.669,Z 446.405,A -85,B 0,C 180,E1 -19819.045,E2 -19819.045} C_VEL
LIN {X 0,Y 259.476,Z 442.728,A -85,B 0,C 180,E1 -19820.485,E2 -19820.485} C_VEL
LIN {X 0,Y 257.358,Z 439.28,A -85,B 0,C 180,E1 -19822.036,E2 -19822.036} C_VEL
LIN {X 0,Y 254.883,Z 435.395,A -85,B 0,C 180,E1 -19824.189,E2 -19824.189} C_VEL
LIN {X 0,Y 252.044,Z 431.283,A -85,B 0,C 180,E1 -19827.542,E2 -19827.542} C_VEL
LIN {X 0,Y 250.631,Z 429.826,A -85,B 0,C 180,E1 -19830.023,E2 -19830.023} C_VEL
LIN {X 0,Y 249.921,Z 429.074,A -85,B 0,C 180,E1 -19832.48,E2 -19832.48} C_VEL
LIN {X 0,Y 249.918,Z 429.125,A -85,B 0,C 180,E1 -19835.366,E2 -19835.366} C_VEL
LIN {X 0,Y 251.045,Z 430.571,A -85,B 0,C 180,E1 -19838.733,E2 -19838.733} C_VEL
LIN {X 0,Y 252.25,Z 431.904,A -85,B 0,C 180,E1 -19840.625,E2 -19840.625} C_VEL
LIN {X 0,Y 254.57,Z 435.606,A -85,B 0,C 180,E1 -19843.379,E2 -19843.379} C_VEL
LIN {X 0,Y 255.678,Z 437.226,A -85,B 0,C 180,E1 -19844.387,E2 -19844.387} C_VEL
LIN {X 0,Y 258.612,Z 441.839,A -85,B 0,C 180,E1 -19846.728,E2 -19846.728} C_VEL
LIN {X 0,Y 260.741,Z 445.518,A -85,B 0,C 180,E1 -19848.204,E2 -19848.204} C_VEL
LIN {X 0,Y 263.048,Z 449.557,A -85,B 0,C 180,E1 -19849.613,E2 -19849.613} C_VEL
LIN {X 0,Y 265.426,Z 454.046,A -85,B 0,C 180,E1 -19850.947,E2 -19850.947} C_VEL
LIN {X 0,Y 267.537,Z 461.929,A -85,B 0,C 180,E1 -19852.353,E2 -19852.353} C_VEL
LIN {X 0,Y 267.845,Z 471.546,A -85,B 0,C 180,E1 -19853.175,E2 -19853.175} C_VEL
LIN {X 0,Y 261.99,Z 523.567,A -85,B 0,C 180,E1 -19855.25,E2 -19855.25} C_VEL
LIN {X 0,Y 259.509,Z 537.444,A -85,B 0,C 180,E1 -19856.046,E2 -19856.046} C_VEL
LIN {X 0,Y 256.586,Z 549.68,A -85,B 0,C 180,E1 -19857.02,E2 -19857.02} C_VEL
LIN {X 0,Y 253.449,Z 560.843,A -85,B 0,C 180,E1 -19858.209,E2 -19858.209} C_VEL
LIN {X 0,Y 249.656,Z 572.375,A -85,B 0,C 180,E1 -19859.791,E2 -19859.791} C_VEL
LIN {X 0,Y 245.375,Z 583.704,A -85,B 0,C 180,E1 -19861.8,E2 -19861.8} C_VEL
LIN {X 0,Y 241.854,Z 592.164,A -85,B 0,C 180,E1 -19863.698,E2 -19863.698} C_VEL
LIN {X 0,Y 238.025,Z 600.725,A -85,B 0,C 180,E1 -19866.154,E2 -19866.154} C_VEL
LIN {X 0,Y 234.447,Z 608.249,A -85,B 0,C 180,E1 -19868.919,E2 -19868.919} C_VEL
LIN {X 0,Y 231.873,Z 613.535,A -85,B 0,C 180,E1 -19871.445,E2 -19871.445} C_VEL
LIN {X 0,Y 229.5,Z 617.69,A -85,B 0,C 180,E1 -19874.004,E2 -19874.004} C_VEL
LIN {X 0,Y 228.357,Z 619.859,A -85,B 0,C 180,E1 -19875.749,E2 -19875.749} C_VEL
LIN {X 0,Y 226.721,Z 622.961,A -85,B 0,C 180,E1 -19879.284,E2 -19879.284} C_VEL
LIN {X 0,Y 226.178,Z 623.899,A -85,B 0,C 180,E1 -19881.064,E2 -19881.064} C_VEL
LIN {X 0,Y 225.688,Z 624.506,A -85,B 0,C 180,E1 -19884.642,E2 -19884.642} C_VEL
LIN {X 0,Y 225.64,Z 624.22,A -85,B 0,C 180,E1 -19886.878,E2 -19886.878} C_VEL
LIN {X 0,Y 225.734,Z 625.891,A -85,B 0,C 180,E1 -19890.002,E2 -19890.002} C_VEL
LIN {X 0,Y 225.656,Z 626.248,A -85,B 0,C 180,E1 -19891.787,E2 -19891.787} C_VEL
LIN {X 0,Y 225.648,Z 625.785,A -85,B 0,C 180,E1 -19895.364,E2 -19895.364} C_VEL
LIN {X 0,Y 225.824,Z 624.955,A -85,B 0,C 180,E1 -19897.153,E2 -19897.153} C_VEL
LIN {X 0,Y 226.653,Z 622.022,A -85,B 0,C 180,E1 -19900.724,E2 -19900.724} C_VEL
LIN {X 0,Y 227.718,Z 618.715,A -85,B 0,C 180,E1 -19903.386,E2 -19903.386} C_VEL
LIN {X 0,Y 229.329,Z 614.356,A -85,B 0,C 180,E1 -19906.013,E2 -19906.013} C_VEL
LIN {X 0,Y 231.831,Z 607.806,A -85,B 0,C 180,E1 -19909.022,E2 -19909.022} C_VEL
LIN {X 0,Y 234.2,Z 600.811,A -85,B 0,C 180,E1 -19911.524,E2 -19911.524} C_VEL
LIN {X 0,Y 237.215,Z 591.827,A -85,B 0,C 180,E1 -19914.042,E2 -19914.042} C_VEL
LIN {X 0,Y 240.487,Z 581.838,A -85,B 0,C 180,E1 -19916.235,E2 -19916.235} C_VEL
LIN {X 0,Y 243.7,Z 570.461,A -85,B 0,C 180,E1 -19918.182,E2 -19918.182} C_VEL
LIN {X 0,Y 246.526,Z 559.08,A -85,B 0,C 180,E1 -19919.694,E2 -19919.694} C_VEL
LIN {X 0,Y 249.208,Z 546.123,A -85,B 0,C 180,E1 -19920.978,E2 -19920.978} C_VEL
LIN {X 0,Y 251.331,Z 533.573,A -85,B 0,C 180,E1 -19921.859,E2 -19921.859} C_VEL
LIN {X 0,Y 252.759,Z 520.629,A -85,B 0,C 180,E1 -19922.492,E2 -19922.492} C_VEL
LIN {X 0,Y 255.73,Z 469.012,A -85,B 0,C 180,E1 -19924.115,E2 -19924.115} C_VEL
LIN {X 0,Y 254.152,Z 456.25,A -85,B 0,C 180,E1 -19924.987,E2 -19924.987} C_VEL
LIN {X 0,Y 249.834,Z 446.027,A -85,B 0,C 180,E1 -19926.392,E2 -19926.392} C_VEL
LIN {X 0,Y 243.872,Z 433.994,A -85,B 0,C 180,E1 -19928.396,E2 -19928.396} C_VEL
LIN {X 0,Y 239.768,Z 426.767,A -85,B 0,C 180,E1 -19929.856,E2 -19929.856} C_VEL
LIN {X 0,Y 237.35,Z 422.766,A -85,B 0,C 180,E1 -19930.752,E2 -19930.752} C_VEL
LIN {X 0,Y 233.987,Z 417.491,A -85,B 0,C 180,E1 -19932.072,E2 -19932.072} C_VEL
LIN {X 0,Y 231.084,Z 413.227,A -85,B 0,C 180,E1 -19933.271,E2 -19933.271} C_VEL
LIN {X 0,Y 230.563,Z 412.048,A -85,B 0,C 180,E1 -19933.584,E2 -19933.584} C_VEL
LIN {X 0,Y 228.916,Z 406.799,A -85,B 0,C 180,E1 -19937.513,E2 -19937.513} C_VEL
LIN {X 0,Y 227.879,Z 403.095,A -85,B 0,C 180,E1 -19940.71,E2 -19940.71} C_VEL
LIN {X 0,Y 227.888,Z 403.097,A -85,B 0,C 180,E1 -19944.13,E2 -19944.13} C_VEL
LIN {X 0,Y 227.877,Z 403.095,A -85,B 0,C 180,E1 -19948.379,E2 -19948.379} C_VEL
LIN {X 0,Y 227.894,Z 403.089,A -85,B 0,C 180,E1 -19952.446,E2 -19952.446} C_VEL
LIN {X 0,Y 227.922,Z 403.086,A -85,B 0,C 180,E1 -19956.368,E2 -19956.368} C_VEL
LIN {X 0,Y 227.95,Z 403.084,A -85,B 0,C 180,E1 -19960.175,E2 -19960.175} C_VEL
LIN {X 0,Y 228.065,Z 403.074,A -85,B 0,C 180,E1 -19963.898,E2 -19963.898} C_VEL
LIN {X 0,Y 228.102,Z 403.073,A -85,B 0,C 180,E1 -19967.545,E2 -19967.545} C_VEL
LIN {X 0,Y 228.314,Z 403.045,A -85,B 0,C 180,E1 -19971.147,E2 -19971.147} C_VEL
LIN {X 0,Y 228.363,Z 403.029,A -85,B 0,C 180,E1 -19972.929,E2 -19972.929} C_VEL
LIN {X 0,Y 228.562,Z 403.009,A -85,B 0,C 180,E1 -19978.238,E2 -19978.238} C_VEL
LIN {X 0,Y 228.562,Z 403.012,A -85,B 0,C 180,E1 -19981.762,E2 -19981.762} C_VEL
LIN {X 0,Y 228.286,Z 403.237,A -85,B 0,C 180,E1 -19985.964,E2 -19985.964} C_VEL
LIN {X 0,Y 229.107,Z 405.536,A -85,B 0,C 180,E1 -19988.046,E2 -19988.046} C_VEL
LIN {X 0,Y 231.253,Z 409.155,A -85,B 0,C 180,E1 -19989.022,E2 -19989.022} C_VEL
LIN {X 0,Y 232.998,Z 411.329,A -85,B 0,C 180,E1 -19989.734,E2 -19989.734} C_VEL
LIN {X 0,Y 236.01,Z 415.645,A -85,B 0,C 180,E1 -19990.933,E2 -19990.933} C_VEL
LIN {X 0,Y 240.616,Z 422.853,A -85,B 0,C 180,E1 -19992.654,E2 -19992.654} C_VEL
LIN {X 0,Y 244.801,Z 429.779,A -85,B 0,C 180,E1 -19994.111,E2 -19994.111} C_VEL
LIN {X 0,Y 248.937,Z 437.439,A -85,B 0,C 180,E1 -19995.486,E2 -19995.486} C_VEL
LIN {X 0,Y 254.308,Z 448.693,A -85,B 0,C 180,E1 -19997.191,E2 -19997.191} C_VEL
LIN {X 0,Y 256.475,Z 454.241,A -85,B 0,C 180,E1 -19997.886,E2 -19997.886} C_VEL
LIN {X 0,Y 252.993,Z 512.063,A -85,B 0,C 180,E1 -19999.71,E2 -19999.71} C_VEL
LIN {X 0,Y 251.572,Z 524.939,A -85,B 0,C 180,E1 -20000.399,E2 -20000.399} C_VEL
LIN {X 0,Y 249.546,Z 537.881,A -85,B 0,C 180,E1 -20001.41,E2 -20001.41} C_VEL
LIN {X 0,Y 247.153,Z 549.956,A -85,B 0,C 180,E1 -20002.72,E2 -20002.72} C_VEL
LIN {X 0,Y 244.575,Z 560.403,A -85,B 0,C 180,E1 -20004.163,E2 -20004.163} C_VEL
LIN {X 0,Y 241.669,Z 570.878,A -85,B 0,C 180,E1 -20006.004,E2 -20006.004} C_VEL
LIN {X 0,Y 238.708,Z 580.266,A -85,B 0,C 180,E1 -20008.104,E2 -20008.104} C_VEL
LIN {X 0,Y 235.75,Z 588.67,A -85,B 0,C 180,E1 -20010.451,E2 -20010.451} C_VEL
LIN {X 0,Y 233.174,Z 595.515,A -85,B 0,C 180,E1 -20012.856,E2 -20012.856} C_VEL
LIN {X 0,Y 231.037,Z 601.026,A -85,B 0,C 180,E1 -20015.308,E2 -20015.308} C_VEL
LIN {X 0,Y 229.35,Z 605.401,A -85,B 0,C 180,E1 -20017.797,E2 -20017.797} C_VEL
LIN {X 0,Y 227.934,Z 608.838,A -85,B 0,C 180,E1 -20020.354,E2 -20020.354} C_VEL
LIN {X 0,Y 226.79,Z 611.375,A -85,B 0,C 180,E1 -20022.982,E2 -20022.982} C_VEL
LIN {X 0,Y 226.01,Z 613.005,A -85,B 0,C 180,E1 -20025.661,E2 -20025.661} C_VEL
LIN {X 0,Y 225.39,Z 613.781,A -85,B 0,C 180,E1 -20029.092,E2 -20029.092} C_VEL
LIN {X 0,Y 225.212,Z 613.451,A -85,B 0,C 180,E1 -20031.38,E2 -20031.38} C_VEL
LIN {X 0,Y 225.286,Z 612.149,A -85,B 0,C 180,E1 -20034.204,E2 -20034.204} C_VEL
LIN {X 0,Y 225.634,Z 609.58,A -85,B 0,C 180,E1 -20037.246,E2 -20037.246} C_VEL
LIN {X 0,Y 226.367,Z 605.587,A -85,B 0,C 180,E1 -20040.38,E2 -20040.38} C_VEL
LIN {X 0,Y 227.378,Z 599.639,A -85,B 0,C 180,E1 -20043.684,E2 -20043.684} C_VEL
LIN {X 0,Y 228.642,Z 593.119,A -85,B 0,C 180,E1 -20046.445,E2 -20046.445} C_VEL
LIN {X 0,Y 230.115,Z 585.622,A -85,B 0,C 180,E1 -20048.968,E2 -20048.968} C_VEL
LIN {X 0,Y 231.993,Z 576.29,A -85,B 0,C 180,E1 -20051.451,E2 -20051.451} C_VEL
LIN {X 0,Y 233.926,Z 566.201,A -85,B 0,C 180,E1 -20053.595,E2 -20053.595} C_VEL
LIN {X 0,Y 235.629,Z 556.131,A -85,B 0,C 180,E1 -20055.312,E2 -20055.312} C_VEL
LIN {X 0,Y 237.317,Z 544.961,A -85,B 0,C 180,E1 -20056.815,E2 -20056.815} C_VEL
LIN {X 0,Y 238.893,Z 532.396,A -85,B 0,C 180,E1 -20058.114,E2 -20058.114} C_VEL
LIN {X 0,Y 240.143,Z 519.324,A -85,B 0,C 180,E1 -20059.085,E2 -20059.085} C_VEL
LIN {X 0,Y 241.001,Z 506.284,A -85,B 0,C 180,E1 -20059.709,E2 -20059.709} C_VEL
LIN {X 0,Y 243.526,Z 442.872,A -85,B 0,C 180,E1 -20061.727,E2 -20061.727} C_VEL
LIN {X 0,Y 234.03,Z 416.936,A -85,B 0,C 180,E1 -20063.739,E2 -20063.739} C_VEL
LIN {X 0,Y 229.579,Z 406.444,A -85,B 0,C 180,E1 -20064.686,E2 -20064.686} C_VEL
LIN {X 0,Y 228.297,Z 403.778,A -85,B 0,C 180,E1 -20064.948,E2 -20064.948} C_VEL
LIN {X 0,Y 228.194,Z 403.06,A -85,B 0,C 180,E1 -20065.029,E2 -20065.029} C_VEL
LIN {X 0,Y 228.557,Z 403.02,A -85,B 0,C 180,E1 -20068.236,E2 -20068.236} C_VEL
LIN {X 0,Y 228.558,Z 403.017,A -85,B 0,C 180,E1 -20071.76,E2 -20071.76} C_VEL
LIN {X 0,Y 228.361,Z 403.034,A -85,B 0,C 180,E1 -20077.069,E2 -20077.069} C_VEL
LIN {X 0,Y 228.173,Z 403.063,A -85,B 0,C 180,E1 -20080.647,E2 -20080.647} C_VEL
LIN {X 0,Y 228.058,Z 403.079,A -85,B 0,C 180,E1 -20086.1,E2 -20086.1} C_VEL
LIN {X 0,Y 227.942,Z 403.083,A -85,B 0,C 180,E1 -20089.823,E2 -20089.823} C_VEL
LIN {X 0,Y 227.912,Z 403.096,A -85,B 0,C 180,E1 -20093.63,E2 -20093.63} C_VEL
LIN {X 0,Y 227.877,Z 403.086,A -85,B 0,C 180,E1 -20097.553,E2 -20097.553} C_VEL
LIN {X 0,Y 227.866,Z 403.1,A -85,B 0,C 180,E1 -20101.62,E2 -20101.62} C_VEL
LIN {X 0,Y 227.898,Z 403.098,A -85,B 0,C 180,E1 -20105.865,E2 -20105.865} C_VEL
LIN {X 0,Y 227.904,Z 403.096,A -85,B 0,C 180,E1 -20108.513,E2 -20108.513} C_VEL
LIN {X 0,Y 233.548,Z 419.683,A -85,B 0,C 180,E1 -20109.71,E2 -20109.71} C_VEL
LIN {X 0,Y 238.422,Z 436.079,A -85,B 0,C 180,E1 -20110.773,E2 -20110.773} C_VEL
LIN {X 0,Y 238.901,Z 439.71,A -85,B 0,C 180,E1 -20110.961,E2 -20110.961} C_VEL
LIN {X 0,Y 235.563,Z 511.062,A -85,B 0,C 180,E1 -20113.859,E2 -20113.859} C_VEL
LIN {X 0,Y 234.755,Z 523.692,A -85,B 0,C 180,E1 -20114.682,E2 -20114.682} C_VEL
LIN {X 0,Y 233.571,Z 537.036,A -85,B 0,C 180,E1 -20115.907,E2 -20115.907} C_VEL
LIN {X 0,Y 232.248,Z 549.169,A -85,B 0,C 180,E1 -20117.383,E2 -20117.383} C_VEL
LIN {X 0,Y 230.857,Z 560.676,A -85,B 0,C 180,E1 -20119.175,E2 -20119.175} C_VEL
LIN {X 0,Y 229.603,Z 570.792,A -85,B 0,C 180,E1 -20121.134,E2 -20121.134} C_VEL
LIN {X 0,Y 228.191,Z 581.107,A -85,B 0,C 180,E1 -20123.631,E2 -20123.631} C_VEL
LIN {X 0,Y 227.207,Z 589.511,A -85,B 0,C 180,E1 -20126.166,E2 -20126.166} C_VEL
LIN {X 0,Y 226.441,Z 596.185,A -85,B 0,C 180,E1 -20128.676,E2 -20128.676} C_VEL
LIN {X 0,Y 225.953,Z 601.828,A -85,B 0,C 180,E1 -20131.337,E2 -20131.337} C_VEL
LIN {X 0,Y 225.501,Z 606.414,A -85,B 0,C 180,E1 -20134.13,E2 -20134.13} C_VEL
LIN {X 0,Y 225.265,Z 608.89,A -85,B 0,C 180,E1 -20136.072,E2 -20136.072} C_VEL
LIN {X 0,Y 225.283,Z 611.819,A -85,B 0,C 180,E1 -20139.364,E2 -20139.364} C_VEL
LIN {X 0,Y 225.539,Z 613.079,A -85,B 0,C 180,E1 -20141.843,E2 -20141.843} C_VEL
LIN {X 0,Y 226.097,Z 613.542,A -85,B 0,C 180,E1 -20144.484,E2 -20144.484} C_VEL
LIN {X 0,Y 227.099,Z 612.958,A -85,B 0,C 180,E1 -20147.489,E2 -20147.489} C_VEL
LIN {X 0,Y 228.321,Z 611.542,A -85,B 0,C 180,E1 -20150.047,E2 -20150.047} C_VEL
LIN {X 0,Y 230.479,Z 608.444,A -85,B 0,C 180,E1 -20153.24,E2 -20153.24} C_VEL
LIN {X 0,Y 232.578,Z 605.035,A -85,B 0,C 180,E1 -20155.665,E2 -20155.665} C_VEL
LIN {X 0,Y 235.353,Z 600.161,A -85,B 0,C 180,E1 -20158.289,E2 -20158.289} C_VEL
LIN {X 0,Y 237.398,Z 596.343,A -85,B 0,C 180,E1 -20159.935,E2 -20159.935} C_VEL
LIN {X 0,Y 238.437,Z 593.452,A -85,B 0,C 180,E1 -20161.152,E2 -20161.152} C_VEL
LIN {X 0,Y 238.606,Z 588.685,A -85,B 0,C 180,E1 -20163.244,E2 -20163.244} C_VEL
LIN {X 0,Y 238.913,Z 583.338,A -85,B 0,C 180,E1 -20165.238,E2 -20165.238} C_VEL
LIN {X 0,Y 240.108,Z 579.546,A -85,B 0,C 180,E1 -20166.275,E2 -20166.275} C_VEL
LIN {X 0,Y 244.497,Z 568.984,A -85,B 0,C 180,E1 -20168.471,E2 -20168.471} C_VEL
LIN {X 0,Y 248.425,Z 558.375,A -85,B 0,C 180,E1 -20170.185,E2 -20170.185} C_VEL
LIN {X 0,Y 251.818,Z 547.512,A -85,B 0,C 180,E1 -20171.583,E2 -20171.583} C_VEL
LIN {X 0,Y 254.895,Z 535.852,A -85,B 0,C 180,E1 -20172.743,E2 -20172.743} C_VEL
LIN {X 0,Y 257.067,Z 525.558,A -85,B 0,C 180,E1 -20173.538,E2 -20173.538} C_VEL
LIN {X 0,Y 259.202,Z 512.585,A -85,B 0,C 180,E1 -20174.266,E2 -20174.266} C_VEL
LIN {X 0,Y 264.826,Z 464.774,A -85,B 0,C 180,E1 -20176.158,E2 -20176.158} C_VEL
LIN {X 0,Y 261.466,Z 457.249,A -85,B 0,C 180,E1 -20178.112,E2 -20178.112} C_VEL
LIN {X 0,Y 258.423,Z 451.206,A -85,B 0,C 180,E1 -20180.096,E2 -20180.096} C_VEL
LIN {X 0,Y 255.109,Z 445.551,A -85,B 0,C 180,E1 -20182.599,E2 -20182.599} C_VEL
LIN {X 0,Y 252.782,Z 441.757,A -85,B 0,C 180,E1 -20184.79,E2 -20184.79} C_VEL
LIN {X 0,Y 250.359,Z 438.034,A -85,B 0,C 180,E1 -20187.892,E2 -20187.892} C_VEL
LIN {X 0,Y 248.878,Z 436.474,A -85,B 0,C 180,E1 -20190.84,E2 -20190.84} C_VEL
LIN {X 0,Y 248.435,Z 435.899,A -85,B 0,C 180,E1 -20194.457,E2 -20194.457} C_VEL
LIN {X 0,Y 249.023,Z 436.847,A -85,B 0,C 180,E1 -20197.358,E2 -20197.358} C_VEL
LIN {X 0,Y 250.521,Z 438.521,A -85,B 0,C 180,E1 -20200.183,E2 -20200.183} C_VEL
LIN {X 0,Y 252.68,Z 442.239,A -85,B 0,C 180,E1 -20202.988,E2 -20202.988} C_VEL
LIN {X 0,Y 253.681,Z 443.792,A -85,B 0,C 180,E1 -20203.969,E2 -20203.969} C_VEL
LIN {X 0,Y 256.198,Z 448,A -85,B 0,C 180,E1 -20206.136,E2 -20206.136} C_VEL
LIN {X 0,Y 259.358,Z 453.524,A -85,B 0,C 180,E1 -20208.377,E2 -20208.377} C_VEL
LIN {X 0,Y 262.18,Z 459.254,A -85,B 0,C 180,E1 -20210.156,E2 -20210.156} C_VEL
LIN {X 0,Y 263.74,Z 465.57,A -85,B 0,C 180,E1 -20211.291,E2 -20211.291} C_VEL
LIN {X 0,Y 263.844,Z 472.921,A -85,B 0,C 180,E1 -20211.94,E2 -20211.94} C_VEL
LIN {X 0,Y 257.773,Z 523.777,A -85,B 0,C 180,E1 -20213.996,E2 -20213.996} C_VEL
LIN {X 0,Y 255.178,Z 537.419,A -85,B 0,C 180,E1 -20214.787,E2 -20214.787} C_VEL
LIN {X 0,Y 251.866,Z 550.355,A -85,B 0,C 180,E1 -20215.839,E2 -20215.839} C_VEL
LIN {X 0,Y 248.565,Z 561.256,A -85,B 0,C 180,E1 -20217.027,E2 -20217.027} C_VEL
LIN {X 0,Y 244.597,Z 572.644,A -85,B 0,C 180,E1 -20218.618,E2 -20218.618} C_VEL
LIN {X 0,Y 240.069,Z 583.86,A -85,B 0,C 180,E1 -20220.639,E2 -20220.639} C_VEL
LIN {X 0,Y 236.354,Z 592.172,A -85,B 0,C 180,E1 -20222.558,E2 -20222.558} C_VEL
LIN {X 0,Y 232.396,Z 600.406,A -85,B 0,C 180,E1 -20224.955,E2 -20224.955} C_VEL
LIN {X 0,Y 228.896,Z 607.138,A -85,B 0,C 180,E1 -20227.433,E2 -20227.433} C_VEL
LIN {X 0,Y 226.102,Z 612.543,A -85,B 0,C 180,E1 -20230.009,E2 -20230.009} C_VEL
LIN {X 0,Y 223.483,Z 616.872,A -85,B 0,C 180,E1 -20232.62,E2 -20232.62} C_VEL
LIN {X 0,Y 221.464,Z 620.138,A -85,B 0,C 180,E1 -20235.296,E2 -20235.296} C_VEL
LIN {X 0,Y 220.509,Z 621.789,A -85,B 0,C 180,E1 -20237.111,E2 -20237.111} C_VEL
LIN {X 0,Y 219.725,Z 623.014,A -85,B 0,C 180,E1 -20238.938,E2 -20238.938} C_VEL
LIN {X 0,Y 218.797,Z 624.239,A -85,B 0,C 180,E1 -20242.62,E2 -20242.62} C_VEL
LIN {X 0,Y 218.54,Z 624.071,A -85,B 0,C 180,E1 -20245.506,E2 -20245.506} C_VEL
LIN {X 0,Y 218.56,Z 623.864,A -85,B 0,C 180,E1 -20246.777,E2 -20246.777} C_VEL
LIN {X 0,Y 218.648,Z 625.625,A -85,B 0,C 180,E1 -20250.002,E2 -20250.002} C_VEL
LIN {X 0,Y 218.552,Z 626.027,A -85,B 0,C 180,E1 -20251.845,E2 -20251.845} C_VEL
LIN {X 0,Y 218.57,Z 625.635,A -85,B 0,C 180,E1 -20255.538,E2 -20255.538} C_VEL
LIN {X 0,Y 218.763,Z 624.859,A -85,B 0,C 180,E1 -20257.386,E2 -20257.386} C_VEL
LIN {X 0,Y 219.109,Z 623.653,A -85,B 0,C 180,E1 -20259.231,E2 -20259.231} C_VEL
LIN {X 0,Y 219.991,Z 621.087,A -85,B 0,C 180,E1 -20261.987,E2 -20261.987} C_VEL
LIN {X 0,Y 221.256,Z 617.522,A -85,B 0,C 180,E1 -20264.723,E2 -20264.723} C_VEL
LIN {X 0,Y 223.231,Z 612.873,A -85,B 0,C 180,E1 -20267.405,E2 -20267.405} C_VEL
LIN {X 0,Y 225.942,Z 605.888,A -85,B 0,C 180,E1 -20270.486,E2 -20270.486} C_VEL
LIN {X 0,Y 228.646,Z 598.412,A -85,B 0,C 180,E1 -20273.075,E2 -20273.075} C_VEL
LIN {X 0,Y 231.4,Z 590.814,A -85,B 0,C 180,E1 -20275.166,E2 -20275.166} C_VEL
LIN {X 0,Y 234.521,Z 581.658,A -85,B 0,C 180,E1 -20277.196,E2 -20277.196} C_VEL
LIN {X 0,Y 237.902,Z 570.282,A -85,B 0,C 180,E1 -20279.174,E2 -20279.174} C_VEL
LIN {X 0,Y 240.855,Z 558.904,A -85,B 0,C 180,E1 -20280.709,E2 -20280.709} C_VEL
LIN {X 0,Y 243.646,Z 545.964,A -85,B 0,C 180,E1 -20282.01,E2 -20282.01} C_VEL
LIN {X 0,Y 245.945,Z 532.877,A -85,B 0,C 180,E1 -20282.933,E2 -20282.933} C_VEL
LIN {X 0,Y 247.363,Z 520.175,A -85,B 0,C 180,E1 -20283.557,E2 -20283.557} C_VEL
LIN {X 0,Y 250.419,Z 469.938,A -85,B 0,C 180,E1 -20285.176,E2 -20285.176} C_VEL
LIN {X 0,Y 249.13,Z 459.074,A -85,B 0,C 180,E1 -20285.95,E2 -20285.95} C_VEL
LIN {X 0,Y 243.959,Z 447.082,A -85,B 0,C 180,E1 -20287.725,E2 -20287.725} C_VEL
LIN {X 0,Y 239.011,Z 437.181,A -85,B 0,C 180,E1 -20289.523,E2 -20289.523} C_VEL
LIN {X 0,Y 235.874,Z 431.627,A -85,B 0,C 180,E1 -20290.7,E2 -20290.7} C_VEL
LIN {X 0,Y 233.538,Z 427.695,A -85,B 0,C 180,E1 -20291.631,E2 -20291.631} C_VEL
LIN {X 0,Y 230.39,Z 422.661,A -85,B 0,C 180,E1 -20292.936,E2 -20292.936} C_VEL
LIN {X 0,Y 227.574,Z 418.149,A -85,B 0,C 180,E1 -20294.189,E2 -20294.189} C_VEL
LIN {X 0,Y 223.768,Z 412.925,A -85,B 0,C 180,E1 -20295.981,E2 -20295.981} C_VEL
LIN {X 0,Y 223.176,Z 411.599,A -85,B 0,C 180,E1 -20296.413,E2 -20296.413} C_VEL
LIN {X 0,Y 221.695,Z 406.653,A -85,B 0,C 180,E1 -20300.652,E2 -20300.652} C_VEL
LIN {X 0,Y 220.864,Z 403.966,A -85,B 0,C 180,E1 -20303.371,E2 -20303.371} C_VEL
LIN {X 0,Y 220.825,Z 403.973,A -85,B 0,C 180,E1 -20307.245,E2 -20307.245} C_VEL
LIN {X 0,Y 220.844,Z 403.976,A -85,B 0,C 180,E1 -20311.488,E2 -20311.488} C_VEL
LIN {X 0,Y 220.875,Z 403.972,A -85,B 0,C 180,E1 -20315.566,E2 -20315.566} C_VEL
LIN {X 0,Y 220.9,Z 403.97,A -85,B 0,C 180,E1 -20319.515,E2 -20319.515} C_VEL
LIN {X 0,Y 221.024,Z 403.954,A -85,B 0,C 180,E1 -20323.371,E2 -20323.371} C_VEL
LIN {X 0,Y 221.12,Z 403.93,A -85,B 0,C 180,E1 -20329.006,E2 -20329.006} C_VEL
LIN {X 0,Y 221.298,Z 403.91,A -85,B 0,C 180,E1 -20332.702,E2 -20332.702} C_VEL
LIN {X 0,Y 221.52,Z 403.886,A -85,B 0,C 180,E1 -20338.182,E2 -20338.182} C_VEL
LIN {X 0,Y 221.52,Z 403.889,A -85,B 0,C 180,E1 -20341.818,E2 -20341.818} C_VEL
LIN {X 0,Y 221.266,Z 403.969,A -85,B 0,C 180,E1 -20343.187,E2 -20343.187} C_VEL
LIN {X 0,Y 221.825,Z 406.176,A -85,B 0,C 180,E1 -20345.226,E2 -20345.226} C_VEL
LIN {X 0,Y 225.043,Z 410.465,A -85,B 0,C 180,E1 -20346.838,E2 -20346.838} C_VEL
LIN {X 0,Y 226.302,Z 411.836,A -85,B 0,C 180,E1 -20347.414,E2 -20347.414} C_VEL
LIN {X 0,Y 229.101,Z 415.997,A -85,B 0,C 180,E1 -20348.701,E2 -20348.701} C_VEL
LIN {X 0,Y 233.824,Z 423.104,A -85,B 0,C 180,E1 -20350.676,E2 -20350.676} C_VEL
LIN {X 0,Y 238.678,Z 430.82,A -85,B 0,C 180,E1 -20352.536,E2 -20352.536} C_VEL
LIN {X 0,Y 244.035,Z 440.535,A -85,B 0,C 180,E1 -20354.451,E2 -20354.451} C_VEL
LIN {X 0,Y 249.783,Z 452.859,A -85,B 0,C 180,E1 -20356.39,E2 -20356.39} C_VEL
LIN {X 0,Y 251.181,Z 456.165,A -85,B 0,C 180,E1 -20356.849,E2 -20356.849} C_VEL
LIN {X 0,Y 247.578,Z 512.554,A -85,B 0,C 180,E1 -20358.673,E2 -20358.673} C_VEL
LIN {X 0,Y 246.111,Z 525.037,A -85,B 0,C 180,E1 -20359.351,E2 -20359.351} C_VEL
LIN {X 0,Y 244.012,Z 537.902,A -85,B 0,C 180,E1 -20360.368,E2 -20360.368} C_VEL
LIN {X 0,Y 241.798,Z 548.806,A -85,B 0,C 180,E1 -20361.545,E2 -20361.545} C_VEL
LIN {X 0,Y 238.77,Z 560.626,A -85,B 0,C 180,E1 -20363.18,E2 -20363.18} C_VEL
LIN {X 0,Y 235.962,Z 570.326,A -85,B 0,C 180,E1 -20364.901,E2 -20364.901} C_VEL
LIN {X 0,Y 233.048,Z 579.321,A -85,B 0,C 180,E1 -20366.895,E2 -20366.895} C_VEL
LIN {X 0,Y 229.87,Z 587.915,A -85,B 0,C 180,E1 -20369.287,E2 -20369.287} C_VEL
LIN {X 0,Y 227.043,Z 594.943,A -85,B 0,C 180,E1 -20371.751,E2 -20371.751} C_VEL
LIN {X 0,Y 224.721,Z 600.585,A -85,B 0,C 180,E1 -20374.26,E2 -20374.26} C_VEL
LIN {X 0,Y 222.813,Z 605.122,A -85,B 0,C 180,E1 -20376.82,E2 -20376.82} C_VEL
LIN {X 0,Y 220.875,Z 609.555,A -85,B 0,C 180,E1 -20380.21,E2 -20380.21} C_VEL
LIN {X 0,Y 219.808,Z 611.727,A -85,B 0,C 180,E1 -20382.657,E2 -20382.657} C_VEL
LIN {X 0,Y 219.057,Z 613.16,A -85,B 0,C 180,E1 -20385.101,E2 -20385.101} C_VEL
LIN {X 0,Y 218.46,Z 613.922,A -85,B 0,C 180,E1 -20387.725,E2 -20387.725} C_VEL
LIN {X 0,Y 218.159,Z 613.805,A -85,B 0,C 180,E1 -20390.639,E2 -20390.639} C_VEL
LIN {X 0,Y 218.149,Z 612.624,A -85,B 0,C 180,E1 -20393.651,E2 -20393.651} C_VEL
LIN {X 0,Y 218.475,Z 610.157,A -85,B 0,C 180,E1 -20396.845,E2 -20396.845} C_VEL
LIN {X 0,Y 219.144,Z 606.439,A -85,B 0,C 180,E1 -20399.986,E2 -20399.986} C_VEL
LIN {X 0,Y 220.175,Z 600.666,A -85,B 0,C 180,E1 -20403.454,E2 -20403.454} C_VEL
LIN {X 0,Y 221.427,Z 594.391,A -85,B 0,C 180,E1 -20406.282,E2 -20406.282} C_VEL
LIN {X 0,Y 223.108,Z 586.029,A -85,B 0,C 180,E1 -20409.242,E2 -20409.242} C_VEL
LIN {X 0,Y 225.031,Z 576.753,A -85,B 0,C 180,E1 -20411.799,E2 -20411.799} C_VEL
LIN {X 0,Y 226.995,Z 566.95,A -85,B 0,C 180,E1 -20413.957,E2 -20413.957} C_VEL
LIN {X 0,Y 228.814,Z 556.689,A -85,B 0,C 180,E1 -20415.773,E2 -20415.773} C_VEL
LIN {X 0,Y 230.697,Z 544.554,A -85,B 0,C 180,E1 -20417.447,E2 -20417.447} C_VEL
LIN {X 0,Y 232.308,Z 531.954,A -85,B 0,C 180,E1 -20418.767,E2 -20418.767} C_VEL
LIN {X 0,Y 233.588,Z 518.625,A -85,B 0,C 180,E1 -20419.757,E2 -20419.757} C_VEL
LIN {X 0,Y 234.499,Z 505.111,A -85,B 0,C 180,E1 -20420.393,E2 -20420.393} C_VEL
LIN {X 0,Y 237.067,Z 444.6,A -85,B 0,C 180,E1 -20422.357,E2 -20422.357} C_VEL
LIN {X 0,Y 227.738,Z 419.093,A -85,B 0,C 180,E1 -20424.415,E2 -20424.415} C_VEL
LIN {X 0,Y 224.032,Z 410.419,A -85,B 0,C 180,E1 -20425.221,E2 -20425.221} C_VEL
LIN {X 0,Y 221.375,Z 404.944,A -85,B 0,C 180,E1 -20425.787,E2 -20425.787} C_VEL
LIN {X 0,Y 221.169,Z 403.938,A -85,B 0,C 180,E1 -20425.897,E2 -20425.897} C_VEL
LIN {X 0,Y 221.515,Z 403.897,A -85,B 0,C 180,E1 -20428.18,E2 -20428.18} C_VEL
LIN {X 0,Y 221.516,Z 403.895,A -85,B 0,C 180,E1 -20431.816,E2 -20431.816} C_VEL
LIN {X 0,Y 221.314,Z 403.912,A -85,B 0,C 180,E1 -20437.295,E2 -20437.295} C_VEL
LIN {X 0,Y 221.118,Z 403.941,A -85,B 0,C 180,E1 -20440.991,E2 -20440.991} C_VEL
LIN {X 0,Y 221.017,Z 403.953,A -85,B 0,C 180,E1 -20446.627,E2 -20446.627} C_VEL
LIN {X 0,Y 220.891,Z 403.966,A -85,B 0,C 180,E1 -20450.483,E2 -20450.483} C_VEL
LIN {X 0,Y 220.865,Z 403.97,A -85,B 0,C 180,E1 -20454.432,E2 -20454.432} C_VEL
LIN {X 0,Y 220.825,Z 403.967,A -85,B 0,C 180,E1 -20458.512,E2 -20458.512} C_VEL
LIN {X 0,Y 220.82,Z 403.977,A -85,B 0,C 180,E1 -20462.752,E2 -20462.752} C_VEL
LIN {X 0,Y 220.833,Z 403.979,A -85,B 0,C 180,E1 -20467.667,E2 -20467.667} C_VEL
LIN {X 0,Y 220.842,Z 403.977,A -85,B 0,C 180,E1 -20467.951,E2 -20467.951} C_VEL
LIN {X 0,Y 226.726,Z 421.084,A -85,B 0,C 180,E1 -20469.247,E2 -20469.247} C_VEL
LIN {X 0,Y 231.733,Z 437.807,A -85,B 0,C 180,E1 -20470.377,E2 -20470.377} C_VEL
LIN {X 0,Y 232.06,Z 440.463,A -85,B 0,C 180,E1 -20470.518,E2 -20470.518} C_VEL
LIN {X 0,Y 228.621,Z 511.499,A -85,B 0,C 180,E1 -20473.506,E2 -20473.506} C_VEL
LIN {X 0,Y 227.823,Z 523.76,A -85,B 0,C 180,E1 -20474.332,E2 -20474.332} C_VEL
LIN {X 0,Y 226.562,Z 537.353,A -85,B 0,C 180,E1 -20475.617,E2 -20475.617} C_VEL
LIN {X 0,Y 225.349,Z 548.382,A -85,B 0,C 180,E1 -20476.982,E2 -20476.982} C_VEL
LIN {X 0,Y 223.873,Z 560.371,A -85,B 0,C 180,E1 -20478.884,E2 -20478.884} C_VEL
LIN {X 0,Y 222.599,Z 570.273,A -85,B 0,C 180,E1 -20480.842,E2 -20480.842} C_VEL
LIN {X 0,Y 221.165,Z 580.741,A -85,B 0,C 180,E1 -20483.428,E2 -20483.428} C_VEL
LIN {X 0,Y 220.11,Z 589.435,A -85,B 0,C 180,E1 -20486.111,E2 -20486.111} C_VEL
LIN {X 0,Y 219.26,Z 597.145,A -85,B 0,C 180,E1 -20489.146,E2 -20489.146} C_VEL
LIN {X 0,Y 218.675,Z 603.239,A -85,B 0,C 180,E1 -20492.224,E2 -20492.224} C_VEL
LIN {X 0,Y 218.243,Z 607.693,A -85,B 0,C 180,E1 -20495.251,E2 -20495.251} C_VEL
LIN {X 0,Y 218.095,Z 609.928,A -85,B 0,C 180,E1 -20497.251,E2 -20497.251} C_VEL
LIN {X 0,Y 218.169,Z 611.641,A -85,B 0,C 180,E1 -20499.246,E2 -20499.246} C_VEL
LIN {X 0,Y 218.346,Z 612.81,A -85,B 0,C 180,E1 -20501.223,E2 -20501.223} C_VEL
LIN {X 0,Y 218.958,Z 613.715,A -85,B 0,C 180,E1 -20504.338,E2 -20504.338} C_VEL
LIN {X 0,Y 219.792,Z 613.542,A -85,B 0,C 180,E1 -20507.066,E2 -20507.066} C_VEL
LIN {X 0,Y 221.184,Z 612.31,A -85,B 0,C 180,E1 -20510.05,E2 -20510.05} C_VEL
LIN {X 0,Y 223.674,Z 609.251,A -85,B 0,C 180,E1 -20513.686,E2 -20513.686} C_VEL
LIN {X 0,Y 226.123,Z 605.662,A -85,B 0,C 180,E1 -20516.436,E2 -20516.436} C_VEL
LIN {X 0,Y 229.077,Z 600.881,A -85,B 0,C 180,E1 -20519.121,E2 -20519.121} C_VEL
LIN {X 0,Y 232.555,Z 594.78,A -85,B 0,C 180,E1 -20521.732,E2 -20521.732} C_VEL
LIN {X 0,Y 236.476,Z 587.226,A -85,B 0,C 180,E1 -20524.261,E2 -20524.261} C_VEL
LIN {X 0,Y 240.108,Z 579.546,A -85,B 0,C 180,E1 -20526.275,E2 -20526.275} C_VEL
LIN {X 0,Y 241.393,Z 575.608,A -85,B 0,C 180,E1 -20527.275,E2 -20527.275} C_VEL
LIN {X 0,Y 242.162,Z 569.249,A -85,B 0,C 180,E1 -20529.071,E2 -20529.071} C_VEL
LIN {X 0,Y 242.912,Z 562.504,A -85,B 0,C 180,E1 -20530.764,E2 -20530.764} C_VEL
LIN {X 0,Y 244.103,Z 557.927,A -85,B 0,C 180,E1 -20531.586,E2 -20531.586} C_VEL
LIN {X 0,Y 247.632,Z 547.205,A -85,B 0,C 180,E1 -20532.953,E2 -20532.953} C_VEL
LIN {X 0,Y 250.802,Z 535.762,A -85,B 0,C 180,E1 -20534.09,E2 -20534.09} C_VEL
LIN {X 0,Y 253.454,Z 523.721,A -85,B 0,C 180,E1 -20534.988,E2 -20534.988} C_VEL
LIN {X 0,Y 255.657,Z 510.381,A -85,B 0,C 180,E1 -20535.692,E2 -20535.692} C_VEL
LIN {X 0,Y 260.859,Z 468.196,A -85,B 0,C 180,E1 -20537.362,E2 -20537.362} C_VEL
LIN {X 0,Y 257.167,Z 459.776,A -85,B 0,C 180,E1 -20539.791,E2 -20539.791} C_VEL
LIN {X 0,Y 254.79,Z 455.301,A -85,B 0,C 180,E1 -20541.531,E2 -20541.531} C_VEL
LIN {X 0,Y 252.651,Z 451.444,A -85,B 0,C 180,E1 -20543.376,E2 -20543.376} C_VEL
LIN {X 0,Y 250.967,Z 448.474,A -85,B 0,C 180,E1 -20545.126,E2 -20545.126} C_VEL
LIN {X 0,Y 248.676,Z 444.774,A -85,B 0,C 180,E1 -20548.248,E2 -20548.248} C_VEL
LIN {X 0,Y 247.281,Z 443.186,A -85,B 0,C 180,E1 -20551.506,E2 -20551.506} C_VEL
LIN {X 0,Y 247.067,Z 442.977,A -85,B 0,C 180,E1 -20555.118,E2 -20555.118} C_VEL
LIN {X 0,Y 247.955,Z 444.303,A -85,B 0,C 180,E1 -20558.304,E2 -20558.304} C_VEL
LIN {X 0,Y 248.915,Z 445.45,A -85,B 0,C 180,E1 -20559.966,E2 -20559.966} C_VEL
LIN {X 0,Y 250.927,Z 449.004,A -85,B 0,C 180,E1 -20562.704,E2 -20562.704} C_VEL
LIN {X 0,Y 251.787,Z 450.619,A -85,B 0,C 180,E1 -20563.653,E2 -20563.653} C_VEL
LIN {X 0,Y 253.918,Z 454.272,A -85,B 0,C 180,E1 -20565.601,E2 -20565.601} C_VEL
LIN {X 0,Y 256.767,Z 459.586,A -85,B 0,C 180,E1 -20567.776,E2 -20567.776} C_VEL
LIN {X 0,Y 259.138,Z 464.582,A -85,B 0,C 180,E1 -20569.368,E2 -20569.368} C_VEL
LIN {X 0,Y 260.023,Z 469.193,A -85,B 0,C 180,E1 -20570.186,E2 -20570.186} C_VEL
LIN {X 0,Y 259.992,Z 474.686,A -85,B 0,C 180,E1 -20570.668,E2 -20570.668} C_VEL
LIN {X 0,Y 253.929,Z 522.803,A -85,B 0,C 180,E1 -20572.618,E2 -20572.618} C_VEL
LIN {X 0,Y 251.261,Z 536.393,A -85,B 0,C 180,E1 -20573.41,E2 -20573.41} C_VEL
LIN {X 0,Y 247.792,Z 549.493,A -85,B 0,C 180,E1 -20574.452,E2 -20574.452} C_VEL
LIN {X 0,Y 244.295,Z 560.545,A -85,B 0,C 180,E1 -20575.63,E2 -20575.63} C_VEL
LIN {X 0,Y 240.125,Z 571.942,A -85,B 0,C 180,E1 -20577.22,E2 -20577.22} C_VEL
LIN {X 0,Y 235.712,Z 582.21,A -85,B 0,C 180,E1 -20579.05,E2 -20579.05} C_VEL
LIN {X 0,Y 230.964,Z 592.314,A -85,B 0,C 180,E1 -20581.366,E2 -20581.366} C_VEL
LIN {X 0,Y 226.739,Z 600.438,A -85,B 0,C 180,E1 -20583.791,E2 -20583.791} C_VEL
LIN {X 0,Y 222.428,Z 608.091,A -85,B 0,C 180,E1 -20586.739,E2 -20586.739} C_VEL
LIN {X 0,Y 219.48,Z 613.269,A -85,B 0,C 180,E1 -20589.379,E2 -20589.379} C_VEL
LIN {X 0,Y 216.74,Z 617.355,A -85,B 0,C 180,E1 -20592.061,E2 -20592.061} C_VEL
LIN {X 0,Y 214.588,Z 620.426,A -85,B 0,C 180,E1 -20594.813,E2 -20594.813} C_VEL
LIN {X 0,Y 212.749,Z 623.034,A -85,B 0,C 180,E1 -20598.571,E2 -20598.571} C_VEL
LIN {X 0,Y 211.729,Z 624.079,A -85,B 0,C 180,E1 -20602.373,E2 -20602.373} C_VEL
LIN {X 0,Y 211.473,Z 623.69,A -85,B 0,C 180,E1 -20605.568,E2 -20605.568} C_VEL
LIN {X 0,Y 211.456,Z 623.409,A -85,B 0,C 180,E1 -20606.565,E2 -20606.565} C_VEL
LIN {X 0,Y 211.563,Z 625.33,A -85,B 0,C 180,E1 -20610.002,E2 -20610.002} C_VEL
LIN {X 0,Y 211.452,Z 625.803,A -85,B 0,C 180,E1 -20611.907,E2 -20611.907} C_VEL
LIN {X 0,Y 211.42,Z 625.792,A -85,B 0,C 180,E1 -20614.244,E2 -20614.244} C_VEL
LIN {X 0,Y 211.692,Z 624.75,A -85,B 0,C 180,E1 -20617.634,E2 -20617.634} C_VEL
LIN {X 0,Y 212.084,Z 623.616,A -85,B 0,C 180,E1 -20619.54,E2 -20619.54} C_VEL
LIN {X 0,Y 212.684,Z 622.035,A -85,B 0,C 180,E1 -20621.438,E2 -20621.438} C_VEL
LIN {X 0,Y 213.87,Z 618.89,A -85,B 0,C 180,E1 -20624.27,E2 -20624.27} C_VEL
LIN {X 0,Y 215.701,Z 614.719,A -85,B 0,C 180,E1 -20627.054,E2 -20627.054} C_VEL
LIN {X 0,Y 218.44,Z 608.386,A -85,B 0,C 180,E1 -20630.237,E2 -20630.237} C_VEL
LIN {X 0,Y 221.091,Z 601.669,A -85,B 0,C 180,E1 -20632.87,E2 -20632.87} C_VEL
LIN {X 0,Y 224.401,Z 593.072,A -85,B 0,C 180,E1 -20635.51,E2 -20635.51} C_VEL
LIN {X 0,Y 227.6,Z 584.397,A -85,B 0,C 180,E1 -20637.595,E2 -20637.595} C_VEL
LIN {X 0,Y 231.069,Z 573.808,A -85,B 0,C 180,E1 -20639.622,E2 -20639.622} C_VEL
LIN {X 0,Y 234.077,Z 563.406,A -85,B 0,C 180,E1 -20641.195,E2 -20641.195} C_VEL
LIN {X 0,Y 236.929,Z 551.964,A -85,B 0,C 180,E1 -20642.525,E2 -20642.525} C_VEL
LIN {X 0,Y 239.293,Z 540.326,A -85,B 0,C 180,E1 -20643.542,E2 -20643.542} C_VEL
LIN {X 0,Y 241.442,Z 526.55,A -85,B 0,C 180,E1 -20644.385,E2 -20644.385} C_VEL
LIN {X 0,Y 242.608,Z 512.395,A -85,B 0,C 180,E1 -20644.95,E2 -20644.95} C_VEL
LIN {X 0,Y 245.214,Z 470.971,A -85,B 0,C 180,E1 -20646.285,E2 -20646.285} C_VEL
LIN {X 0,Y 244.232,Z 462.188,A -85,B 0,C 180,E1 -20646.928,E2 -20646.928} C_VEL
LIN {X 0,Y 238.818,Z 449.501,A -85,B 0,C 180,E1 -20648.933,E2 -20648.933} C_VEL
LIN {X 0,Y 233.988,Z 439.881,A -85,B 0,C 180,E1 -20650.806,E2 -20650.806} C_VEL
LIN {X 0,Y 230.205,Z 433.175,A -85,B 0,C 180,E1 -20652.377,E2 -20652.377} C_VEL
LIN {X 0,Y 227.059,Z 428.112,A -85,B 0,C 180,E1 -20653.743,E2 -20653.743} C_VEL
LIN {X 0,Y 223.645,Z 422.727,A -85,B 0,C 180,E1 -20655.365,E2 -20655.365} C_VEL
LIN {X 0,Y 220.624,Z 418.19,A -85,B 0,C 180,E1 -20656.902,E2 -20656.902} C_VEL
LIN {X 0,Y 216.3,Z 412.35,A -85,B 0,C 180,E1 -20659.335,E2 -20659.335} C_VEL
LIN {X 0,Y 215.753,Z 411.147,A -85,B 0,C 180,E1 -20659.807,E2 -20659.807} C_VEL
LIN {X 0,Y 214.538,Z 407.204,A -85,B 0,C 180,E1 -20663.867,E2 -20663.867} C_VEL
LIN {X 0,Y 213.79,Z 404.846,A -85,B 0,C 180,E1 -20666.871,E2 -20666.871} C_VEL
LIN {X 0,Y 213.788,Z 404.845,A -85,B 0,C 180,E1 -20670.455,E2 -20670.455} C_VEL
LIN {X 0,Y 213.809,Z 404.847,A -85,B 0,C 180,E1 -20674.703,E2 -20674.703} C_VEL
LIN {X 0,Y 213.821,Z 404.847,A -85,B 0,C 180,E1 -20678.804,E2 -20678.804} C_VEL
LIN {X 0,Y 213.952,Z 404.829,A -85,B 0,C 180,E1 -20682.804,E2 -20682.804} C_VEL
LIN {X 0,Y 213.988,Z 404.823,A -85,B 0,C 180,E1 -20686.709,E2 -20686.709} C_VEL
LIN {X 0,Y 214.176,Z 404.799,A -85,B 0,C 180,E1 -20690.557,E2 -20690.557} C_VEL
LIN {X 0,Y 214.236,Z 404.791,A -85,B 0,C 180,E1 -20692.46,E2 -20692.46} C_VEL
LIN {X 0,Y 214.483,Z 404.769,A -85,B 0,C 180,E1 -20699.061,E2 -20699.061} C_VEL
LIN {X 0,Y 214.554,Z 404.775,A -85,B 0,C 180,E1 -20700,E2 -20700} C_VEL
LIN {X 0,Y 214.872,Z 406.482,A -85,B 0,C 180,E1 -20701.933,E2 -20701.933} C_VEL
LIN {X 0,Y 216.167,Z 408.805,A -85,B 0,C 180,E1 -20702.795,E2 -20702.795} C_VEL
LIN {X 0,Y 219.721,Z 413.069,A -85,B 0,C 180,E1 -20704.811,E2 -20704.811} C_VEL
LIN {X 0,Y 223.563,Z 418.054,A -85,B 0,C 180,E1 -20706.77,E2 -20706.77} C_VEL
LIN {X 0,Y 227.304,Z 423.747,A -85,B 0,C 180,E1 -20708.554,E2 -20708.554} C_VEL
LIN {X 0,Y 230.468,Z 428.553,A -85,B 0,C 180,E1 -20709.919,E2 -20709.919} C_VEL
LIN {X 0,Y 235.214,Z 436.449,A -85,B 0,C 180,E1 -20711.853,E2 -20711.853} C_VEL
LIN {X 0,Y 240.035,Z 445.386,A -85,B 0,C 180,E1 -20713.66,E2 -20713.66} C_VEL
LIN {X 0,Y 245.412,Z 457.352,A -85,B 0,C 180,E1 -20715.603,E2 -20715.603} C_VEL
LIN {X 0,Y 245.96,Z 458.69,A -85,B 0,C 180,E1 -20715.794,E2 -20715.794} C_VEL
LIN {X 0,Y 242.308,Z 512.807,A -85,B 0,C 180,E1 -20717.563,E2 -20717.563} C_VEL
LIN {X 0,Y 240.742,Z 525.54,A -85,B 0,C 180,E1 -20718.266,E2 -20718.266} C_VEL
LIN {X 0,Y 238.774,Z 537.275,A -85,B 0,C 180,E1 -20719.204,E2 -20719.204} C_VEL
LIN {X 0,Y 236.386,Z 548.507,A -85,B 0,C 180,E1 -20720.408,E2 -20720.408} C_VEL
LIN {X 0,Y 233.341,Z 559.977,A -85,B 0,C 180,E1 -20722.005,E2 -20722.005} C_VEL
LIN {X 0,Y 229.929,Z 571.068,A -85,B 0,C 180,E1 -20723.997,E2 -20723.997} C_VEL
LIN {X 0,Y 226.852,Z 579.992,A -85,B 0,C 180,E1 -20726.043,E2 -20726.043} C_VEL
LIN {X 0,Y 223.665,Z 588.164,A -85,B 0,C 180,E1 -20728.376,E2 -20728.376} C_VEL
LIN {X 0,Y 220.82,Z 594.841,A -85,B 0,C 180,E1 -20730.755,E2 -20730.755} C_VEL
LIN {X 0,Y 217.895,Z 601.554,A -85,B 0,C 180,E1 -20733.842,E2 -20733.842} C_VEL
LIN {X 0,Y 215.534,Z 606.673,A -85,B 0,C 180,E1 -20737.014,E2 -20737.014} C_VEL
LIN {X 0,Y 214.037,Z 609.805,A -85,B 0,C 180,E1 -20739.633,E2 -20739.633} C_VEL
LIN {X 0,Y 213.291,Z 611.265,A -85,B 0,C 180,E1 -20741.225,E2 -20741.225} C_VEL
LIN {X 0,Y 212.251,Z 613.123,A -85,B 0,C 180,E1 -20744.055,E2 -20744.055} C_VEL
LIN {X 0,Y 211.488,Z 614.078,A -85,B 0,C 180,E1 -20746.978,E2 -20746.978} C_VEL
LIN {X 0,Y 211.067,Z 613.906,A -85,B 0,C 180,E1 -20750.751,E2 -20750.751} C_VEL
LIN {X 0,Y 211.014,Z 613.003,A -85,B 0,C 180,E1 -20753.163,E2 -20753.163} C_VEL
LIN {X 0,Y 211.273,Z 610.849,A -85,B 0,C 180,E1 -20756.267,E2 -20756.267} C_VEL
LIN {X 0,Y 211.941,Z 607.268,A -85,B 0,C 180,E1 -20759.561,E2 -20759.561} C_VEL
LIN {X 0,Y 212.91,Z 601.929,A -85,B 0,C 180,E1 -20763.032,E2 -20763.032} C_VEL
LIN {X 0,Y 214.231,Z 595.353,A -85,B 0,C 180,E1 -20766.222,E2 -20766.222} C_VEL
LIN {X 0,Y 215.763,Z 587.983,A -85,B 0,C 180,E1 -20769.002,E2 -20769.002} C_VEL
LIN {X 0,Y 217.679,Z 579.173,A -85,B 0,C 180,E1 -20771.65,E2 -20771.65} C_VEL
LIN {X 0,Y 219.685,Z 569.531,A -85,B 0,C 180,E1 -20773.954,E2 -20773.954} C_VEL
LIN {X 0,Y 221.734,Z 558.674,A -85,B 0,C 180,E1 -20776.012,E2 -20776.012} C_VEL
LIN {X 0,Y 223.714,Z 546.975,A -85,B 0,C 180,E1 -20777.755,E2 -20777.755} C_VEL
LIN {X 0,Y 225.305,Z 535.201,A -85,B 0,C 180,E1 -20779.097,E2 -20779.097} C_VEL
LIN {X 0,Y 226.742,Z 521.454,A -85,B 0,C 180,E1 -20780.243,E2 -20780.243} C_VEL
LIN {X 0,Y 227.784,Z 508.742,A -85,B 0,C 180,E1 -20780.927,E2 -20780.927} C_VEL
LIN {X 0,Y 230.577,Z 446.174,A -85,B 0,C 180,E1 -20783.032,E2 -20783.032} C_VEL
LIN {X 0,Y 221.281,Z 420.706,A -85,B 0,C 180,E1 -20785.159,E2 -20785.159} C_VEL
LIN {X 0,Y 218.012,Z 413.484,A -85,B 0,C 180,E1 -20785.885,E2 -20785.885} C_VEL
LIN {X 0,Y 214.387,Z 405.792,A -85,B 0,C 180,E1 -20786.709,E2 -20786.709} C_VEL
LIN {X 0,Y 214.219,Z 404.801,A -85,B 0,C 180,E1 -20786.824,E2 -20786.824} C_VEL
LIN {X 0,Y 214.553,Z 404.758,A -85,B 0,C 180,E1 -20789.998,E2 -20789.998} C_VEL
LIN {X 0,Y 214.45,Z 404.774,A -85,B 0,C 180,E1 -20791.876,E2 -20791.876} C_VEL
LIN {X 0,Y 214.25,Z 404.791,A -85,B 0,C 180,E1 -20797.537,E2 -20797.537} C_VEL
LIN {X 0,Y 214.049,Z 404.821,A -85,B 0,C 180,E1 -20801.359,E2 -20801.359} C_VEL
LIN {X 0,Y 213.934,Z 404.837,A -85,B 0,C 180,E1 -20805.234,E2 -20805.234} C_VEL
LIN {X 0,Y 213.839,Z 404.838,A -85,B 0,C 180,E1 -20809.185,E2 -20809.185} C_VEL
LIN {X 0,Y 213.846,Z 404.847,A -85,B 0,C 180,E1 -20813.224,E2 -20813.224} C_VEL
LIN {X 0,Y 213.827,Z 404.835,A -85,B 0,C 180,E1 -20817.447,E2 -20817.447} C_VEL
LIN {X 0,Y 213.767,Z 404.857,A -85,B 0,C 180,E1 -20821.734,E2 -20821.734} C_VEL
LIN {X 0,Y 213.755,Z 404.858,A -85,B 0,C 180,E1 -20826.283,E2 -20826.283} C_VEL
LIN {X 0,Y 213.814,Z 404.883,A -85,B 0,C 180,E1 -20827.425,E2 -20827.425} C_VEL
LIN {X 0,Y 220.212,Z 423.445,A -85,B 0,C 180,E1 -20828.849,E2 -20828.849} C_VEL
LIN {X 0,Y 225.093,Z 439.752,A -85,B 0,C 180,E1 -20829.978,E2 -20829.978} C_VEL
LIN {X 0,Y 223.709,Z 471.115,A -85,B 0,C 180,E1 -20831.33,E2 -20831.33} C_VEL
LIN {X 0,Y 221.71,Z 511.139,A -85,B 0,C 180,E1 -20833.107,E2 -20833.107} C_VEL
LIN {X 0,Y 220.806,Z 524.453,A -85,B 0,C 180,E1 -20834.037,E2 -20834.037} C_VEL
LIN {X 0,Y 219.513,Z 538.056,A -85,B 0,C 180,E1 -20835.383,E2 -20835.383} C_VEL
LIN {X 0,Y 218.034,Z 550.848,A -85,B 0,C 180,E1 -20837.083,E2 -20837.083} C_VEL
LIN {X 0,Y 216.636,Z 562.182,A -85,B 0,C 180,E1 -20839.005,E2 -20839.005} C_VEL
LIN {X 0,Y 215.147,Z 573.056,A -85,B 0,C 180,E1 -20841.337,E2 -20841.337} C_VEL
LIN {X 0,Y 213.922,Z 582.167,A -85,B 0,C 180,E1 -20843.746,E2 -20843.746} C_VEL
LIN {X 0,Y 212.901,Z 590.347,A -85,B 0,C 180,E1 -20846.431,E2 -20846.431} C_VEL
LIN {X 0,Y 212.075,Z 597.776,A -85,B 0,C 180,E1 -20849.493,E2 -20849.493} C_VEL
LIN {X 0,Y 211.57,Z 603.116,A -85,B 0,C 180,E1 -20852.286,E2 -20852.286} C_VEL
LIN {X 0,Y 211.152,Z 607.663,A -85,B 0,C 180,E1 -20855.414,E2 -20855.414} C_VEL
LIN {X 0,Y 211.047,Z 611.104,A -85,B 0,C 180,E1 -20858.807,E2 -20858.807} C_VEL
LIN {X 0,Y 211.456,Z 613.374,A -85,B 0,C 180,E1 -20862.595,E2 -20862.595} C_VEL
LIN {X 0,Y 211.921,Z 613.881,A -85,B 0,C 180,E1 -20864.615,E2 -20864.615} C_VEL
LIN {X 0,Y 212.498,Z 613.958,A -85,B 0,C 180,E1 -20866.614,E2 -20866.614} C_VEL
LIN {X 0,Y 214.047,Z 613.036,A -85,B 0,C 180,E1 -20870.053,E2 -20870.053} C_VEL
LIN {X 0,Y 215.583,Z 611.496,A -85,B 0,C 180,E1 -20872.507,E2 -20872.507} C_VEL
LIN {X 0,Y 218.416,Z 608.103,A -85,B 0,C 180,E1 -20875.9,E2 -20875.9} C_VEL
LIN {X 0,Y 221.737,Z 603.328,A -85,B 0,C 180,E1 -20879.092,E2 -20879.092} C_VEL
LIN {X 0,Y 225.3,Z 597.846,A -85,B 0,C 180,E1 -20881.787,E2 -20881.787} C_VEL
LIN {X 0,Y 229.268,Z 590.976,A -85,B 0,C 180,E1 -20884.395,E2 -20884.395} C_VEL
LIN {X 0,Y 233.799,Z 582.31,A -85,B 0,C 180,E1 -20886.906,E2 -20886.906} C_VEL
LIN {X 0,Y 237.921,Z 573.544,A -85,B 0,C 180,E1 -20888.921,E2 -20888.921} C_VEL
LIN {X 0,Y 241.888,Z 563.945,A -85,B 0,C 180,E1 -20890.675,E2 -20890.675} C_VEL
LIN {X 0,Y 244.103,Z 557.927,A -85,B 0,C 180,E1 -20891.586,E2 -20891.586} C_VEL
LIN {X 0,Y 245.306,Z 553.191,A -85,B 0,C 180,E1 -20892.369,E2 -20892.369} C_VEL
LIN {X 0,Y 246.079,Z 545.568,A -85,B 0,C 180,E1 -20893.841,E2 -20893.841} C_VEL
LIN {X 0,Y 246.753,Z 537.63,A -85,B 0,C 180,E1 -20895.189,E2 -20895.189} C_VEL
LIN {X 0,Y 247.732,Z 532.415,A -85,B 0,C 180,E1 -20895.769,E2 -20895.769} C_VEL
LIN {X 0,Y 250.736,Z 518.313,A -85,B 0,C 180,E1 -20896.701,E2 -20896.701} C_VEL
LIN {X 0,Y 253.092,Z 502.337,A -85,B 0,C 180,E1 -20897.397,E2 -20897.397} C_VEL
LIN {X 0,Y 257.036,Z 471.65,A -85,B 0,C 180,E1 -20898.633,E2 -20898.633} C_VEL
LIN {X 0,Y 253.811,Z 464.101,A -85,B 0,C 180,E1 -20901.02,E2 -20901.02} C_VEL
LIN {X 0,Y 252.308,Z 461.195,A -85,B 0,C 180,E1 -20902.264,E2 -20902.264} C_VEL
LIN {X 0,Y 250.566,Z 457.864,A -85,B 0,C 180,E1 -20903.88,E2 -20903.88} C_VEL
LIN {X 0,Y 249.045,Z 455.043,A -85,B 0,C 180,E1 -20905.587,E2 -20905.587} C_VEL
LIN {X 0,Y 247.007,Z 451.547,A -85,B 0,C 180,E1 -20908.609,E2 -20908.609} C_VEL
LIN {X 0,Y 245.762,Z 450.002,A -85,B 0,C 180,E1 -20912.011,E2 -20912.011} C_VEL
LIN {X 0,Y 245.67,Z 449.983,A -85,B 0,C 180,E1 -20915.348,E2 -20915.348} C_VEL
LIN {X 0,Y 246.91,Z 451.728,A -85,B 0,C 180,E1 -20919.033,E2 -20919.033} C_VEL
LIN {X 0,Y 247.452,Z 452.772,A -85,B 0,C 180,E1 -20920.031,E2 -20920.031} C_VEL
LIN {X 0,Y 249.61,Z 456.633,A -85,B 0,C 180,E1 -20922.945,E2 -20922.945} C_VEL
LIN {X 0,Y 251.888,Z 460.93,A -85,B 0,C 180,E1 -20925.215,E2 -20925.215} C_VEL
LIN {X 0,Y 254.694,Z 466.608,A -85,B 0,C 180,E1 -20927.498,E2 -20927.498} C_VEL
LIN {X 0,Y 256.104,Z 469.993,A -85,B 0,C 180,E1 -20928.556,E2 -20928.556} C_VEL
LIN {X 0,Y 256.555,Z 472.846,A -85,B 0,C 180,E1 -20929.044,E2 -20929.044} C_VEL
LIN {X 0,Y 256.411,Z 476.453,A -85,B 0,C 180,E1 -20929.337,E2 -20929.337} C_VEL
LIN {X 0,Y 250.149,Z 522.955,A -85,B 0,C 180,E1 -20931.248,E2 -20931.248} C_VEL
LIN {X 0,Y 247.251,Z 537.023,A -85,B 0,C 180,E1 -20932.074,E2 -20932.074} C_VEL
LIN {X 0,Y 243.917,Z 548.956,A -85,B 0,C 180,E1 -20933.028,E2 -20933.028} C_VEL
LIN {X 0,Y 240.215,Z 559.971,A -85,B 0,C 180,E1 -20934.19,E2 -20934.19} C_VEL
LIN {X 0,Y 235.816,Z 571.351,A -85,B 0,C 180,E1 -20935.772,E2 -20935.772} C_VEL
LIN {X 0,Y 230.729,Z 582.63,A -85,B 0,C 180,E1 -20937.791,E2 -20937.791} C_VEL
LIN {X 0,Y 226.509,Z 591.019,A -85,B 0,C 180,E1 -20939.725,E2 -20939.725} C_VEL
LIN {X 0,Y 221.904,Z 599.314,A -85,B 0,C 180,E1 -20942.153,E2 -20942.153} C_VEL
LIN {X 0,Y 217.134,Z 607.135,A -85,B 0,C 180,E1 -20945.12,E2 -20945.12} C_VEL
LIN {X 0,Y 213.877,Z 612.41,A -85,B 0,C 180,E1 -20947.8,E2 -20947.8} C_VEL
LIN {X 0,Y 210.92,Z 616.62,A -85,B 0,C 180,E1 -20950.539,E2 -20950.539} C_VEL
LIN {X 0,Y 209.158,Z 618.879,A -85,B 0,C 180,E1 -20952.4,E2 -20952.4} C_VEL
LIN {X 0,Y 207.727,Z 620.665,A -85,B 0,C 180,E1 -20954.299,E2 -20954.299} C_VEL
LIN {X 0,Y 205.788,Z 623.058,A -85,B 0,C 180,E1 -20958.179,E2 -20958.179} C_VEL
LIN {X 0,Y 205.115,Z 623.667,A -85,B 0,C 180,E1 -20960.138,E2 -20960.138} C_VEL
LIN {X 0,Y 204.469,Z 623.64,A -85,B 0,C 180,E1 -20964.084,E2 -20964.084} C_VEL
LIN {X 0,Y 204.38,Z 623.031,A -85,B 0,C 180,E1 -20966.448,E2 -20966.448} C_VEL
LIN {X 0,Y 204.48,Z 625.03,A -85,B 0,C 180,E1 -20970.003,E2 -20970.003} C_VEL
LIN {X 0,Y 204.355,Z 625.557,A -85,B 0,C 180,E1 -20971.973,E2 -20971.973} C_VEL
LIN {X 0,Y 204.322,Z 625.644,A -85,B 0,C 180,E1 -20974.047,E2 -20974.047} C_VEL
LIN {X 0,Y 204.645,Z 624.641,A -85,B 0,C 180,E1 -20977.898,E2 -20977.898} C_VEL
LIN {X 0,Y 205.077,Z 623.559,A -85,B 0,C 180,E1 -20979.869,E2 -20979.869} C_VEL
LIN {X 0,Y 205.707,Z 622.058,A -85,B 0,C 180,E1 -20981.831,E2 -20981.831} C_VEL
LIN {X 0,Y 206.968,Z 619.011,A -85,B 0,C 180,E1 -20984.757,E2 -20984.757} C_VEL
LIN {X 0,Y 208.915,Z 614.931,A -85,B 0,C 180,E1 -20987.626,E2 -20987.626} C_VEL
LIN {X 0,Y 211.792,Z 608.708,A -85,B 0,C 180,E1 -20990.901,E2 -20990.901} C_VEL
LIN {X 0,Y 214.633,Z 601.979,A -85,B 0,C 180,E1 -20993.65,E2 -20993.65} C_VEL
LIN {X 0,Y 218.064,Z 593.708,A -85,B 0,C 180,E1 -20996.307,E2 -20996.307} C_VEL
LIN {X 0,Y 221.375,Z 585.274,A -85,B 0,C 180,E1 -20998.44,E2 -20998.44} C_VEL
LIN {X 0,Y 225.004,Z 574.938,A -85,B 0,C 180,E1 -21000.504,E2 -21000.504} C_VEL
LIN {X 0,Y 228.521,Z 563.414,A -85,B 0,C 180,E1 -21002.303,E2 -21002.303} C_VEL
LIN {X 0,Y 231.494,Z 552.053,A -85,B 0,C 180,E1 -21003.648,E2 -21003.648} C_VEL
LIN {X 0,Y 234.178,Z 539.266,A -85,B 0,C 180,E1 -21004.768,E2 -21004.768} C_VEL
LIN {X 0,Y 236.347,Z 525.739,A -85,B 0,C 180,E1 -21005.579,E2 -21005.579} C_VEL
LIN {X 0,Y 237.64,Z 509.522,A -85,B 0,C 180,E1 -21006.214,E2 -21006.214} C_VEL
LIN {X 0,Y 240.185,Z 472.366,A -85,B 0,C 180,E1 -21007.419,E2 -21007.419} C_VEL
LIN {X 0,Y 239.373,Z 465.066,A -85,B 0,C 180,E1 -21007.992,E2 -21007.992} C_VEL
LIN {X 0,Y 234.414,Z 453.333,A -85,B 0,C 180,E1 -21009.941,E2 -21009.941} C_VEL
LIN {X 0,Y 229.544,Z 443.264,A -85,B 0,C 180,E1 -21011.997,E2 -21011.997} C_VEL
LIN {X 0,Y 224.232,Z 434.109,A -85,B 0,C 180,E1 -21014.388,E2 -21014.388} C_VEL
LIN {X 0,Y 220.529,Z 428.222,A -85,B 0,C 180,E1 -21016.229,E2 -21016.229} C_VEL
LIN {X 0,Y 217.189,Z 423.151,A -85,B 0,C 180,E1 -21018.056,E2 -21018.056} C_VEL
LIN {X 0,Y 213.585,Z 417.964,A -85,B 0,C 180,E1 -21020.239,E2 -21020.239} C_VEL
LIN {X 0,Y 208.921,Z 411.79,A -85,B 0,C 180,E1 -21023.55,E2 -21023.55} C_VEL
LIN {X 0,Y 208.407,Z 410.724,A -85,B 0,C 180,E1 -21024.035,E2 -21024.035} C_VEL
LIN {X 0,Y 207.339,Z 407.865,A -85,B 0,C 180,E1 -21027.935,E2 -21027.935} C_VEL
LIN {X 0,Y 206.755,Z 405.731,A -85,B 0,C 180,E1 -21031.583,E2 -21031.583} C_VEL
LIN {X 0,Y 206.793,Z 405.715,A -85,B 0,C 180,E1 -21036.585,E2 -21036.585} C_VEL
LIN {X 0,Y 206.881,Z 405.704,A -85,B 0,C 180,E1 -21042.197,E2 -21042.197} C_VEL
LIN {X 0,Y 206.922,Z 405.699,A -85,B 0,C 180,E1 -21046.246,E2 -21046.246} C_VEL
LIN {X 0,Y 207.114,Z 405.676,A -85,B 0,C 180,E1 -21050.232,E2 -21050.232} C_VEL
LIN {X 0,Y 207.176,Z 405.672,A -85,B 0,C 180,E1 -21052.202,E2 -21052.202} C_VEL
LIN {X 0,Y 207.105,Z 405.805,A -85,B 0,C 180,E1 -21055.377,E2 -21055.377} C_VEL
LIN {X 0,Y 207.659,Z 407.199,A -85,B 0,C 180,E1 -21057.576,E2 -21057.576} C_VEL
LIN {X 0,Y 209.566,Z 409.882,A -85,B 0,C 180,E1 -21059.159,E2 -21059.159} C_VEL
LIN {X 0,Y 212.485,Z 412.694,A -85,B 0,C 180,E1 -21061.179,E2 -21061.179} C_VEL
LIN {X 0,Y 215.025,Z 416.644,A -85,B 0,C 180,E1 -21062.869,E2 -21062.869} C_VEL
LIN {X 0,Y 217.385,Z 419.433,A -85,B 0,C 180,E1 -21064.23,E2 -21064.23} C_VEL
LIN {X 0,Y 220.783,Z 424.049,A -85,B 0,C 180,E1 -21066.067,E2 -21066.067} C_VEL
LIN {X 0,Y 224.523,Z 429.903,A -85,B 0,C 180,E1 -21067.927,E2 -21067.927} C_VEL
LIN {X 0,Y 227.338,Z 434.315,A -85,B 0,C 180,E1 -21069.222,E2 -21069.222} C_VEL
LIN {X 0,Y 232.108,Z 442.518,A -85,B 0,C 180,E1 -21071.252,E2 -21071.252} C_VEL
LIN {X 0,Y 236.382,Z 450.882,A -85,B 0,C 180,E1 -21072.962,E2 -21072.962} C_VEL
LIN {X 0,Y 240.806,Z 460.937,A -85,B 0,C 180,E1 -21074.648,E2 -21074.648} C_VEL
LIN {X 0,Y 237.141,Z 512.995,A -85,B 0,C 180,E1 -21076.4,E2 -21076.4} C_VEL
LIN {X 0,Y 235.481,Z 525.984,A -85,B 0,C 180,E1 -21077.129,E2 -21077.129} C_VEL
LIN {X 0,Y 233.375,Z 537.905,A -85,B 0,C 180,E1 -21078.098,E2 -21078.098} C_VEL
LIN {X 0,Y 230.874,Z 549.037,A -85,B 0,C 180,E1 -21079.318,E2 -21079.318} C_VEL
LIN {X 0,Y 227.659,Z 560.561,A -85,B 0,C 180,E1 -21080.953,E2 -21080.953} C_VEL
LIN {X 0,Y 224.175,Z 571.363,A -85,B 0,C 180,E1 -21082.934,E2 -21082.934} C_VEL
LIN {X 0,Y 220.54,Z 581.211,A -85,B 0,C 180,E1 -21085.275,E2 -21085.275} C_VEL
LIN {X 0,Y 216.833,Z 590.08,A -85,B 0,C 180,E1 -21087.962,E2 -21087.962} C_VEL
LIN {X 0,Y 214.154,Z 595.886,A -85,B 0,C 180,E1 -21090.178,E2 -21090.178} C_VEL
LIN {X 0,Y 211.604,Z 601.335,A -85,B 0,C 180,E1 -21092.769,E2 -21092.769} C_VEL
LIN {X 0,Y 208.937,Z 606.771,A -85,B 0,C 180,E1 -21096.165,E2 -21096.165} C_VEL
LIN {X 0,Y 207.338,Z 609.831,A -85,B 0,C 180,E1 -21098.771,E2 -21098.771} C_VEL
LIN {X 0,Y 206.1,Z 612.049,A -85,B 0,C 180,E1 -21101.389,E2 -21101.389} C_VEL
LIN {X 0,Y 205.153,Z 613.525,A -85,B 0,C 180,E1 -21103.991,E2 -21103.991} C_VEL
LIN {X 0,Y 204.482,Z 614.289,A -85,B 0,C 180,E1 -21106.573,E2 -21106.573} C_VEL
LIN {X 0,Y 204.065,Z 614.328,A -85,B 0,C 180,E1 -21109.261,E2 -21109.261} C_VEL
LIN {X 0,Y 203.918,Z 613.437,A -85,B 0,C 180,E1 -21112.438,E2 -21112.438} C_VEL
LIN {X 0,Y 204.116,Z 611.403,A -85,B 0,C 180,E1 -21115.727,E2 -21115.727} C_VEL
LIN {X 0,Y 204.73,Z 608.059,A -85,B 0,C 180,E1 -21119.116,E2 -21119.116} C_VEL
LIN {X 0,Y 205.672,Z 602.966,A -85,B 0,C 180,E1 -21122.679,E2 -21122.679} C_VEL
LIN {X 0,Y 206.93,Z 596.713,A -85,B 0,C 180,E1 -21125.946,E2 -21125.946} C_VEL
LIN {X 0,Y 208.4,Z 589.98,A -85,B 0,C 180,E1 -21128.706,E2 -21128.706} C_VEL
LIN {X 0,Y 210.326,Z 581.411,A -85,B 0,C 180,E1 -21131.489,E2 -21131.489} C_VEL
LIN {X 0,Y 212.241,Z 572.549,A -85,B 0,C 180,E1 -21133.8,E2 -21133.8} C_VEL
LIN {X 0,Y 214.361,Z 562.021,A -85,B 0,C 180,E1 -21136.005,E2 -21136.005} C_VEL
LIN {X 0,Y 216.296,Z 551.202,A -85,B 0,C 180,E1 -21137.792,E2 -21137.792} C_VEL
LIN {X 0,Y 218.15,Z 539.237,A -85,B 0,C 180,E1 -21139.322,E2 -21139.322} C_VEL
LIN {X 0,Y 219.717,Z 526.296,A -85,B 0,C 180,E1 -21140.563,E2 -21140.563} C_VEL
LIN {X 0,Y 220.932,Z 512.613,A -85,B 0,C 180,E1 -21141.441,E2 -21141.441} C_VEL
LIN {X 0,Y 222.152,Z 488.51,A -85,B 0,C 180,E1 -21142.338,E2 -21142.338} C_VEL
LIN {X 0,Y 224.017,Z 447.487,A -85,B 0,C 180,E1 -21143.743,E2 -21143.743} C_VEL
LIN {X 0,Y 215.065,Z 422.962,A -85,B 0,C 180,E1 -21145.89,E2 -21145.89} C_VEL
LIN {X 0,Y 210.763,Z 413.805,A -85,B 0,C 180,E1 -21146.886,E2 -21146.886} C_VEL
LIN {X 0,Y 207.495,Z 406.605,A -85,B 0,C 180,E1 -21147.674,E2 -21147.674} C_VEL
LIN {X 0,Y 207.32,Z 405.664,A -85,B 0,C 180,E1 -21147.782,E2 -21147.782} C_VEL
LIN {X 0,Y 207.518,Z 405.635,A -85,B 0,C 180,E1 -21149.997,E2 -21149.997} C_VEL
LIN {X 0,Y 207.386,Z 405.653,A -85,B 0,C 180,E1 -21151.939,E2 -21151.939} C_VEL
LIN {X 0,Y 207.191,Z 405.671,A -85,B 0,C 180,E1 -21157.795,E2 -21157.795} C_VEL
LIN {X 0,Y 206.984,Z 405.699,A -85,B 0,C 180,E1 -21161.752,E2 -21161.752} C_VEL
LIN {X 0,Y 206.868,Z 405.719,A -85,B 0,C 180,E1 -21165.768,E2 -21165.768} C_VEL
LIN {X 0,Y 206.783,Z 405.717,A -85,B 0,C 180,E1 -21169.866,E2 -21169.866} C_VEL
LIN {X 0,Y 206.762,Z 405.728,A -85,B 0,C 180,E1 -21174.069,E2 -21174.069} C_VEL
LIN {X 0,Y 206.734,Z 405.719,A -85,B 0,C 180,E1 -21178.417,E2 -21178.417} C_VEL
LIN {X 0,Y 206.703,Z 405.736,A -85,B 0,C 180,E1 -21182.954,E2 -21182.954} C_VEL
LIN {X 0,Y 206.736,Z 405.735,A -85,B 0,C 180,E1 -21186.841,E2 -21186.841} C_VEL
LIN {X 0,Y 213.565,Z 425.332,A -85,B 0,C 180,E1 -21188.417,E2 -21188.417} C_VEL
LIN {X 0,Y 218.333,Z 441.179,A -85,B 0,C 180,E1 -21189.555,E2 -21189.555} C_VEL
LIN {X 0,Y 214.757,Z 511,A -85,B 0,C 180,E1 -21192.719,E2 -21192.719} C_VEL
LIN {X 0,Y 213.837,Z 524.564,A -85,B 0,C 180,E1 -21193.692,E2 -21193.692} C_VEL
LIN {X 0,Y 212.566,Z 537.748,A -85,B 0,C 180,E1 -21195.031,E2 -21195.031} C_VEL
LIN {X 0,Y 211.136,Z 549.879,A -85,B 0,C 180,E1 -21196.661,E2 -21196.661} C_VEL
LIN {X 0,Y 209.553,Z 562.433,A -85,B 0,C 180,E1 -21198.838,E2 -21198.838} C_VEL
LIN {X 0,Y 208.132,Z 572.603,A -85,B 0,C 180,E1 -21201.074,E2 -21201.074} C_VEL
LIN {X 0,Y 206.889,Z 581.687,A -85,B 0,C 180,E1 -21203.525,E2 -21203.525} C_VEL
LIN {X 0,Y 205.848,Z 590.03,A -85,B 0,C 180,E1 -21206.302,E2 -21206.302} C_VEL
LIN {X 0,Y 204.958,Z 597.83,A -85,B 0,C 180,E1 -21209.617,E2 -21209.617} C_VEL
LIN {X 0,Y 204.487,Z 602.92,A -85,B 0,C 180,E1 -21212.357,E2 -21212.357} C_VEL
LIN {X 0,Y 204.04,Z 607.573,A -85,B 0,C 180,E1 -21215.585,E2 -21215.585} C_VEL
LIN {X 0,Y 203.935,Z 610.634,A -85,B 0,C 180,E1 -21218.5,E2 -21218.5} C_VEL
LIN {X 0,Y 204.24,Z 613.013,A -85,B 0,C 180,E1 -21221.959,E2 -21221.959} C_VEL
LIN {X 0,Y 204.686,Z 613.823,A -85,B 0,C 180,E1 -21224.057,E2 -21224.057} C_VEL
LIN {X 0,Y 205.238,Z 614.201,A -85,B 0,C 180,E1 -21226.131,E2 -21226.131} C_VEL
LIN {X 0,Y 206.012,Z 614.108,A -85,B 0,C 180,E1 -21228.189,E2 -21228.189} C_VEL
LIN {X 0,Y 206.983,Z 613.567,A -85,B 0,C 180,E1 -21230.225,E2 -21230.225} C_VEL
LIN {X 0,Y 208.212,Z 612.607,A -85,B 0,C 180,E1 -21232.24,E2 -21232.24} C_VEL
LIN {X 0,Y 209.727,Z 611.171,A -85,B 0,C 180,E1 -21234.23,E2 -21234.23} C_VEL
LIN {X 0,Y 212.374,Z 608.188,A -85,B 0,C 180,E1 -21237.155,E2 -21237.155} C_VEL
LIN {X 0,Y 215.529,Z 604.095,A -85,B 0,C 180,E1 -21240,E2 -21240} C_VEL
LIN {X 0,Y 219.973,Z 597.714,A -85,B 0,C 180,E1 -21243.205,E2 -21243.205} C_VEL
LIN {X 0,Y 224.254,Z 590.782,A -85,B 0,C 180,E1 -21245.846,E2 -21245.846} C_VEL
LIN {X 0,Y 229.242,Z 581.833,A -85,B 0,C 180,E1 -21248.438,E2 -21248.438} C_VEL
LIN {X 0,Y 233.912,Z 572.204,A -85,B 0,C 180,E1 -21250.605,E2 -21250.605} C_VEL
LIN {X 0,Y 238.818,Z 560.85,A -85,B 0,C 180,E1 -21252.565,E2 -21252.565} C_VEL
LIN {X 0,Y 242.722,Z 549.978,A -85,B 0,C 180,E1 -21254.034,E2 -21254.034} C_VEL
LIN {X 0,Y 246.377,Z 537.771,A -85,B 0,C 180,E1 -21255.3,E2 -21255.3} C_VEL
LIN {X 0,Y 247.732,Z 532.415,A -85,B 0,C 180,E1 -21255.769,E2 -21255.769} C_VEL
LIN {X 0,Y 248.655,Z 527.053,A -85,B 0,C 180,E1 -21256.31,E2 -21256.31} C_VEL
LIN {X 0,Y 248.948,Z 518.387,A -85,B 0,C 180,E1 -21257.429,E2 -21257.429} C_VEL
LIN {X 0,Y 249.051,Z 509.527,A -85,B 0,C 180,E1 -21258.426,E2 -21258.426} C_VEL
LIN {X 0,Y 249.561,Z 503.88,A -85,B 0,C 180,E1 -21258.773,E2 -21258.773} C_VEL
LIN {X 0,Y 253.489,Z 475.46,A -85,B 0,C 180,E1 -21259.913,E2 -21259.913} C_VEL
LIN {X 0,Y 251.169,Z 469.65,A -85,B 0,C 180,E1 -21261.854,E2 -21261.854} C_VEL
LIN {X 0,Y 248.551,Z 464.297,A -85,B 0,C 180,E1 -21264.387,E2 -21264.387} C_VEL
LIN {X 0,Y 246.973,Z 461.349,A -85,B 0,C 180,E1 -21266.277,E2 -21266.277} C_VEL
LIN {X 0,Y 245.443,Z 458.396,A -85,B 0,C 180,E1 -21268.845,E2 -21268.845} C_VEL
LIN {X 0,Y 244.426,Z 457.114,A -85,B 0,C 180,E1 -21271.517,E2 -21271.517} C_VEL
LIN {X 0,Y 244.125,Z 456.78,A -85,B 0,C 180,E1 -21273.403,E2 -21273.403} C_VEL
LIN {X 0,Y 244.436,Z 457.257,A -85,B 0,C 180,E1 -21276.389,E2 -21276.389} C_VEL
LIN {X 0,Y 245.67,Z 459.129,A -85,B 0,C 180,E1 -21279.434,E2 -21279.434} C_VEL
LIN {X 0,Y 247.141,Z 462.128,A -85,B 0,C 180,E1 -21281.788,E2 -21281.788} C_VEL
LIN {X 0,Y 249.564,Z 466.936,A -85,B 0,C 180,E1 -21284.525,E2 -21284.525} C_VEL
LIN {X 0,Y 252.119,Z 472.541,A -85,B 0,C 180,E1 -21286.82,E2 -21286.82} C_VEL
LIN {X 0,Y 253.136,Z 475.187,A -85,B 0,C 180,E1 -21287.666,E2 -21287.666} C_VEL
LIN {X 0,Y 253.214,Z 476.901,A -85,B 0,C 180,E1 -21287.901,E2 -21287.901} C_VEL
LIN {X 0,Y 246.855,Z 522.193,A -85,B 0,C 180,E1 -21289.769,E2 -21289.769} C_VEL
LIN {X 0,Y 244.02,Z 535.547,A -85,B 0,C 180,E1 -21290.552,E2 -21290.552} C_VEL
LIN {X 0,Y 240.8,Z 546.829,A -85,B 0,C 180,E1 -21291.405,E2 -21291.405} C_VEL
LIN {X 0,Y 236.315,Z 559.59,A -85,B 0,C 180,E1 -21292.706,E2 -21292.706} C_VEL
LIN {X 0,Y 231.716,Z 571.004,A -85,B 0,C 180,E1 -21294.281,E2 -21294.281} C_VEL
LIN {X 0,Y 226.829,Z 581.268,A -85,B 0,C 180,E1 -21296.106,E2 -21296.106} C_VEL
LIN {X 0,Y 221.428,Z 591.354,A -85,B 0,C 180,E1 -21298.422,E2 -21298.422} C_VEL
LIN {X 0,Y 216.537,Z 599.529,A -85,B 0,C 180,E1 -21300.87,E2 -21300.87} C_VEL
LIN {X 0,Y 211.692,Z 606.895,A -85,B 0,C 180,E1 -21303.746,E2 -21303.746} C_VEL
LIN {X 0,Y 208.431,Z 611.617,A -85,B 0,C 180,E1 -21306.135,E2 -21306.135} C_VEL
LIN {X 0,Y 205.304,Z 615.916,A -85,B 0,C 180,E1 -21308.937,E2 -21308.937} C_VEL
LIN {X 0,Y 202.425,Z 619.218,A -85,B 0,C 180,E1 -21311.795,E2 -21311.795} C_VEL
LIN {X 0,Y 200.887,Z 620.903,A -85,B 0,C 180,E1 -21313.75,E2 -21313.75} C_VEL
LIN {X 0,Y 199.734,Z 622.189,A -85,B 0,C 180,E1 -21315.744,E2 -21315.744} C_VEL
LIN {X 0,Y 198.094,Z 623.514,A -85,B 0,C 180,E1 -21319.785,E2 -21319.785} C_VEL
LIN {X 0,Y 197.389,Z 623.304,A -85,B 0,C 180,E1 -21323.871,E2 -21323.871} C_VEL
LIN {X 0,Y 197.312,Z 622.58,A -85,B 0,C 180,E1 -21326.221,E2 -21326.221} C_VEL
LIN {X 0,Y 197.398,Z 624.728,A -85,B 0,C 180,E1 -21330.003,E2 -21330.003} C_VEL
LIN {X 0,Y 197.244,Z 625.458,A -85,B 0,C 180,E1 -21333.911,E2 -21333.911} C_VEL
LIN {X 0,Y 197.343,Z 625.199,A -85,B 0,C 180,E1 -21336.136,E2 -21336.136} C_VEL
LIN {X 0,Y 198.054,Z 623.505,A -85,B 0,C 180,E1 -21340.222,E2 -21340.222} C_VEL
LIN {X 0,Y 198.725,Z 622.075,A -85,B 0,C 180,E1 -21342.253,E2 -21342.253} C_VEL
LIN {X 0,Y 200.091,Z 619.099,A -85,B 0,C 180,E1 -21345.276,E2 -21345.276} C_VEL
LIN {X 0,Y 202.156,Z 615.108,A -85,B 0,C 180,E1 -21348.236,E2 -21348.236} C_VEL
LIN {X 0,Y 204.756,Z 610.025,A -85,B 0,C 180,E1 -21351.127,E2 -21351.127} C_VEL
LIN {X 0,Y 207.619,Z 603.707,A -85,B 0,C 180,E1 -21353.969,E2 -21353.969} C_VEL
LIN {X 0,Y 211.129,Z 595.846,A -85,B 0,C 180,E1 -21356.707,E2 -21356.707} C_VEL
LIN {X 0,Y 215.207,Z 586.11,A -85,B 0,C 180,E1 -21359.333,E2 -21359.333} C_VEL
LIN {X 0,Y 219.009,Z 576.066,A -85,B 0,C 180,E1 -21361.433,E2 -21361.433} C_VEL
LIN {X 0,Y 222.647,Z 564.822,A -85,B 0,C 180,E1 -21363.263,E2 -21363.263} C_VEL
LIN {X 0,Y 225.717,Z 553.954,A -85,B 0,C 180,E1 -21364.63,E2 -21364.63} C_VEL
LIN {X 0,Y 228.485,Z 542.06,A -85,B 0,C 180,E1 -21365.765,E2 -21365.765} C_VEL
LIN {X 0,Y 230.829,Z 529.034,A -85,B 0,C 180,E1 -21366.627,E2 -21366.627} C_VEL
LIN {X 0,Y 232.283,Z 515.61,A -85,B 0,C 180,E1 -21367.24,E2 -21367.24} C_VEL
LIN {X 0,Y 235.267,Z 473.316,A -85,B 0,C 180,E1 -21368.648,E2 -21368.648} C_VEL
LIN {X 0,Y 234.743,Z 468.298,A -85,B 0,C 180,E1 -21369.052,E2 -21369.052} C_VEL
LIN {X 0,Y 229.739,Z 456.254,A -85,B 0,C 180,E1 -21371.175,E2 -21371.175} C_VEL
LIN {X 0,Y 225.458,Z 447.49,A -85,B 0,C 180,E1 -21373.094,E2 -21373.094} C_VEL
LIN {X 0,Y 221.209,Z 439.792,A -85,B 0,C 180,E1 -21375.164,E2 -21375.164} C_VEL
LIN {X 0,Y 217.531,Z 433.805,A -85,B 0,C 180,E1 -21377.088,E2 -21377.088} C_VEL
LIN {X 0,Y 214.543,Z 429.101,A -85,B 0,C 180,E1 -21378.842,E2 -21378.842} C_VEL
LIN {X 0,Y 210.333,Z 422.907,A -85,B 0,C 180,E1 -21381.592,E2 -21381.592} C_VEL
LIN {X 0,Y 206.92,Z 418.196,A -85,B 0,C 180,E1 -21384.214,E2 -21384.214} C_VEL
LIN {X 0,Y 206.277,Z 417.123,A -85,B 0,C 180,E1 -21384.785,E2 -21384.785} C_VEL
LIN {X 0,Y 200.994,Z 410.363,A -85,B 0,C 180,E1 -21390.475,E2 -21390.475} C_VEL
LIN {X 0,Y 200.778,Z 409.796,A -85,B 0,C 180,E1 -21391.061,E2 -21391.061} C_VEL
LIN {X 0,Y 200,Z 407.844,A -85,B 0,C 180,E1 -21396.019,E2 -21396.019} C_VEL
LIN {X 0,Y 199.835,Z 406.698,A -85,B 0,C 180,E1 -21401.732,E2 -21401.732} C_VEL
LIN {X 0,Y 199.876,Z 406.789,A -85,B 0,C 180,E1 -21405.751,E2 -21405.751} C_VEL
LIN {X 0,Y 200.319,Z 407.753,A -85,B 0,C 180,E1 -21410.662,E2 -21410.662} C_VEL
LIN {X 0,Y 202.061,Z 410.672,A -85,B 0,C 180,E1 -21413.259,E2 -21413.259} C_VEL
LIN {X 0,Y 205.849,Z 413.832,A -85,B 0,C 180,E1 -21417.003,E2 -21417.003} C_VEL
LIN {X 0,Y 208.086,Z 416.799,A -85,B 0,C 180,E1 -21418.912,E2 -21418.912} C_VEL
LIN {X 0,Y 210.384,Z 419.273,A -85,B 0,C 180,E1 -21420.578,E2 -21420.578} C_VEL
LIN {X 0,Y 213.674,Z 424.012,A -85,B 0,C 180,E1 -21422.799,E2 -21422.799} C_VEL
LIN {X 0,Y 218.033,Z 429.998,A -85,B 0,C 180,E1 -21425.332,E2 -21425.332} C_VEL
LIN {X 0,Y 223.468,Z 438.637,A -85,B 0,C 180,E1 -21428.108,E2 -21428.108} C_VEL
LIN {X 0,Y 228.209,Z 447.062,A -85,B 0,C 180,E1 -21430.281,E2 -21430.281} C_VEL
LIN {X 0,Y 232.346,Z 455.424,A -85,B 0,C 180,E1 -21432.057,E2 -21432.057} C_VEL
LIN {X 0,Y 235.843,Z 463.573,A -85,B 0,C 180,E1 -21433.483,E2 -21433.483} C_VEL
LIN {X 0,Y 232.152,Z 513.372,A -85,B 0,C 180,E1 -21435.177,E2 -21435.177} C_VEL
LIN {X 0,Y 230.445,Z 525.964,A -85,B 0,C 180,E1 -21435.887,E2 -21435.887} C_VEL
LIN {X 0,Y 228.166,Z 538.288,A -85,B 0,C 180,E1 -21436.903,E2 -21436.903} C_VEL
LIN {X 0,Y 225.487,Z 549.534,A -85,B 0,C 180,E1 -21438.161,E2 -21438.161} C_VEL
LIN {X 0,Y 221.882,Z 561.753,A -85,B 0,C 180,E1 -21439.949,E2 -21439.949} C_VEL
LIN {X 0,Y 218.362,Z 572.017,A -85,B 0,C 180,E1 -21441.891,E2 -21441.891} C_VEL
LIN {X 0,Y 215.179,Z 580.269,A -85,B 0,C 180,E1 -21443.859,E2 -21443.859} C_VEL
LIN {X 0,Y 211.651,Z 588.436,A -85,B 0,C 180,E1 -21446.287,E2 -21446.287} C_VEL
LIN {X 0,Y 207.827,Z 596.335,A -85,B 0,C 180,E1 -21449.281,E2 -21449.281} C_VEL
LIN {X 0,Y 204.615,Z 602.693,A -85,B 0,C 180,E1 -21452.491,E2 -21452.491} C_VEL
LIN {X 0,Y 202.406,Z 606.818,A -85,B 0,C 180,E1 -21455.219,E2 -21455.219} C_VEL
LIN {X 0,Y 200.638,Z 609.986,A -85,B 0,C 180,E1 -21457.986,E2 -21457.986} C_VEL
LIN {X 0,Y 198.662,Z 613.164,A -85,B 0,C 180,E1 -21462.234,E2 -21462.234} C_VEL
LIN {X 0,Y 197.661,Z 614.335,A -85,B 0,C 180,E1 -21465.326,E2 -21465.326} C_VEL
LIN {X 0,Y 197.05,Z 614.577,A -85,B 0,C 180,E1 -21468.503,E2 -21468.503} C_VEL
LIN {X 0,Y 196.836,Z 613.462,A -85,B 0,C 180,E1 -21472.625,E2 -21472.625} C_VEL
LIN {X 0,Y 197.12,Z 610.924,A -85,B 0,C 180,E1 -21476.45,E2 -21476.45} C_VEL
LIN {X 0,Y 197.861,Z 606.959,A -85,B 0,C 180,E1 -21480.177,E2 -21480.177} C_VEL
LIN {X 0,Y 198.92,Z 601.555,A -85,B 0,C 180,E1 -21483.789,E2 -21483.789} C_VEL
LIN {X 0,Y 200.474,Z 594.425,A -85,B 0,C 180,E1 -21487.315,E2 -21487.315} C_VEL
LIN {X 0,Y 202.242,Z 586.539,A -85,B 0,C 180,E1 -21490.356,E2 -21490.356} C_VEL
LIN {X 0,Y 204.202,Z 578.127,A -85,B 0,C 180,E1 -21492.921,E2 -21492.921} C_VEL
LIN {X 0,Y 206.516,Z 567.663,A -85,B 0,C 180,E1 -21495.462,E2 -21495.462} C_VEL
LIN {X 0,Y 208.682,Z 556.513,A -85,B 0,C 180,E1 -21497.599,E2 -21497.599} C_VEL
LIN {X 0,Y 210.847,Z 543.998,A -85,B 0,C 180,E1 -21499.434,E2 -21499.434} C_VEL
LIN {X 0,Y 212.469,Z 532.39,A -85,B 0,C 180,E1 -21500.732,E2 -21500.732} C_VEL
LIN {X 0,Y 213.827,Z 519.602,A -85,B 0,C 180,E1 -21501.765,E2 -21501.765} C_VEL
LIN {X 0,Y 214.856,Z 505.723,A -85,B 0,C 180,E1 -21502.479,E2 -21502.479} C_VEL
LIN {X 0,Y 217.599,Z 449.2,A -85,B 0,C 180,E1 -21504.466,E2 -21504.466} C_VEL
LIN {X 0,Y 209.145,Z 425.945,A -85,B 0,C 180,E1 -21506.585,E2 -21506.585} C_VEL
LIN {X 0,Y 200.503,Z 407.298,A -85,B 0,C 180,E1 -21508.711,E2 -21508.711} C_VEL
LIN {X 0,Y 200.373,Z 406.527,A -85,B 0,C 180,E1 -21508.867,E2 -21508.867} C_VEL
LIN {X 0,Y 200.326,Z 406.532,A -85,B 0,C 180,E1 -21512.008,E2 -21512.008} C_VEL
LIN {X 0,Y 200.134,Z 406.551,A -85,B 0,C 180,E1 -21518.072,E2 -21518.072} C_VEL
LIN {X 0,Y 199.916,Z 406.577,A -85,B 0,C 180,E1 -21522.174,E2 -21522.174} C_VEL
LIN {X 0,Y 199.805,Z 406.597,A -85,B 0,C 180,E1 -21526.341,E2 -21526.341} C_VEL
LIN {X 0,Y 199.699,Z 406.604,A -85,B 0,C 180,E1 -21530.602,E2 -21530.602} C_VEL
LIN {X 0,Y 199.671,Z 406.609,A -85,B 0,C 180,E1 -21534.981,E2 -21534.981} C_VEL
LIN {X 0,Y 199.662,Z 406.604,A -85,B 0,C 180,E1 -21539.521,E2 -21539.521} C_VEL
LIN {X 0,Y 199.655,Z 406.614,A -85,B 0,C 180,E1 -21542.347,E2 -21542.347} C_VEL
LIN {X 0,Y 199.684,Z 406.611,A -85,B 0,C 180,E1 -21546.209,E2 -21546.209} C_VEL
LIN {X 0,Y 206.831,Z 426.961,A -85,B 0,C 180,E1 -21547.935,E2 -21547.935} C_VEL
LIN {X 0,Y 211.478,Z 442.804,A -85,B 0,C 180,E1 -21549.113,E2 -21549.113} C_VEL
LIN {X 0,Y 207.771,Z 511.395,A -85,B 0,C 180,E1 -21552.335,E2 -21552.335} C_VEL
LIN {X 0,Y 206.885,Z 524.557,A -85,B 0,C 180,E1 -21553.313,E2 -21553.313} C_VEL
LIN {X 0,Y 205.576,Z 537.723,A -85,B 0,C 180,E1 -21554.688,E2 -21554.688} C_VEL
LIN {X 0,Y 204.201,Z 549.303,A -85,B 0,C 180,E1 -21556.278,E2 -21556.278} C_VEL
LIN {X 0,Y 202.621,Z 561.508,A -85,B 0,C 180,E1 -21558.443,E2 -21558.443} C_VEL
LIN {X 0,Y 201.274,Z 571.089,A -85,B 0,C 180,E1 -21560.555,E2 -21560.555} C_VEL
LIN {X 0,Y 199.856,Z 581.07,A -85,B 0,C 180,E1 -21563.286,E2 -21563.286} C_VEL
LIN {X 0,Y 198.794,Z 589.559,A -85,B 0,C 180,E1 -21566.164,E2 -21566.164} C_VEL
LIN {X 0,Y 197.938,Z 596.832,A -85,B 0,C 180,E1 -21569.263,E2 -21569.263} C_VEL
LIN {X 0,Y 197.39,Z 602.699,A -85,B 0,C 180,E1 -21572.428,E2 -21572.428} C_VEL
LIN {X 0,Y 196.933,Z 607.451,A -85,B 0,C 180,E1 -21575.769,E2 -21575.769} C_VEL
LIN {X 0,Y 196.855,Z 610.862,A -85,B 0,C 180,E1 -21579.083,E2 -21579.083} C_VEL
LIN {X 0,Y 197.039,Z 612.448,A -85,B 0,C 180,E1 -21581.276,E2 -21581.276} C_VEL
LIN {X 0,Y 197.514,Z 613.754,A -85,B 0,C 180,E1 -21583.877,E2 -21583.877} C_VEL
LIN {X 0,Y 198.696,Z 614.433,A -85,B 0,C 180,E1 -21587.747,E2 -21587.747} C_VEL
LIN {X 0,Y 199.751,Z 614.148,A -85,B 0,C 180,E1 -21590.094,E2 -21590.094} C_VEL
LIN {X 0,Y 200.859,Z 613.539,A -85,B 0,C 180,E1 -21591.954,E2 -21591.954} C_VEL
LIN {X 0,Y 202.334,Z 612.407,A -85,B 0,C 180,E1 -21594.018,E2 -21594.018} C_VEL
LIN {X 0,Y 204.241,Z 610.672,A -85,B 0,C 180,E1 -21596.238,E2 -21596.238} C_VEL
LIN {X 0,Y 207.041,Z 607.623,A -85,B 0,C 180,E1 -21599.027,E2 -21599.027} C_VEL
LIN {X 0,Y 210.977,Z 602.871,A -85,B 0,C 180,E1 -21602.15,E2 -21602.15} C_VEL
LIN {X 0,Y 215.522,Z 596.621,A -85,B 0,C 180,E1 -21605.145,E2 -21605.145} C_VEL
LIN {X 0,Y 220.42,Z 589.047,A -85,B 0,C 180,E1 -21607.879,E2 -21607.879} C_VEL
LIN {X 0,Y 225.559,Z 580.236,A -85,B 0,C 180,E1 -21610.321,E2 -21610.321} C_VEL
LIN {X 0,Y 230.282,Z 570.909,A -85,B 0,C 180,E1 -21612.335,E2 -21612.335} C_VEL
LIN {X 0,Y 235.334,Z 559.399,A -85,B 0,C 180,E1 -21614.263,E2 -21614.263} C_VEL
LIN {X 0,Y 239.746,Z 547.593,A -85,B 0,C 180,E1 -21615.777,E2 -21615.777} C_VEL
LIN {X 0,Y 243.342,Z 535.782,A -85,B 0,C 180,E1 -21616.936,E2 -21616.936} C_VEL
LIN {X 0,Y 246.242,Z 523.852,A -85,B 0,C 180,E1 -21617.805,E2 -21617.805} C_VEL
LIN {X 0,Y 248.495,Z 511.418,A -85,B 0,C 180,E1 -21618.467,E2 -21618.467} C_VEL
LIN {X 0,Y 249.561,Z 503.88,A -85,B 0,C 180,E1 -21618.773,E2 -21618.773} C_VEL
LIN {X 0,Y 249.819,Z 500.104,A -85,B 0,C 180,E1 -21619.05,E2 -21619.05} C_VEL
LIN {X 0,Y 249.409,Z 494.404,A -85,B 0,C 180,E1 -21619.873,E2 -21619.873} C_VEL
LIN {X 0,Y 249.021,Z 488.715,A -85,B 0,C 180,E1 -21620.714,E2 -21620.714} C_VEL
LIN {X 0,Y 249.279,Z 484.945,A -85,B 0,C 180,E1 -21621.013,E2 -21621.013} C_VEL
LIN {X 0,Y 250.091,Z 479.244,A -85,B 0,C 180,E1 -21621.257,E2 -21621.257} C_VEL
LIN {X 0,Y 248.194,Z 474.323,A -85,B 0,C 180,E1 -21623.094,E2 -21623.094} C_VEL
LIN {X 0,Y 246.43,Z 470.487,A -85,B 0,C 180,E1 -21625.049,E2 -21625.049} C_VEL
LIN {X 0,Y 245.232,Z 468.042,A -85,B 0,C 180,E1 -21626.641,E2 -21626.641} C_VEL
LIN {X 0,Y 243.823,Z 465.146,A -85,B 0,C 180,E1 -21629.219,E2 -21629.219} C_VEL
LIN {X 0,Y 242.886,Z 463.906,A -85,B 0,C 180,E1 -21632.088,E2 -21632.088} C_VEL
LIN {X 0,Y 242.812,Z 463.904,A -85,B 0,C 180,E1 -21635.372,E2 -21635.372} C_VEL
LIN {X 0,Y 243.943,Z 465.691,A -85,B 0,C 180,E1 -21638.938,E2 -21638.938} C_VEL
LIN {X 0,Y 245.751,Z 469.655,A -85,B 0,C 180,E1 -21641.969,E2 -21641.969} C_VEL
LIN {X 0,Y 247.623,Z 473.717,A -85,B 0,C 180,E1 -21644.188,E2 -21644.188} C_VEL
LIN {X 0,Y 249.836,Z 479.045,A -85,B 0,C 180,E1 -21646.344,E2 -21646.344} C_VEL
LIN {X 0,Y 250.069,Z 479.549,A -85,B 0,C 180,E1 -21646.536,E2 -21646.536} C_VEL
LIN {X 0,Y 243.631,Z 522.412,A -85,B 0,C 180,E1 -21648.292,E2 -21648.292} C_VEL
LIN {X 0,Y 240.343,Z 536.724,A -85,B 0,C 180,E1 -21649.138,E2 -21649.138} C_VEL
LIN {X 0,Y 236.732,Z 548.512,A -85,B 0,C 180,E1 -21650.063,E2 -21650.063} C_VEL
LIN {X 0,Y 232.604,Z 559.509,A -85,B 0,C 180,E1 -21651.178,E2 -21651.178} C_VEL
LIN {X 0,Y 227.801,Z 570.76,A -85,B 0,C 180,E1 -21652.741,E2 -21652.741} C_VEL
LIN {X 0,Y 222.142,Z 581.912,A -85,B 0,C 180,E1 -21654.736,E2 -21654.736} C_VEL
LIN {X 0,Y 217.376,Z 590.293,A -85,B 0,C 180,E1 -21656.662,E2 -21656.662} C_VEL
LIN {X 0,Y 212.104,Z 598.584,A -85,B 0,C 180,E1 -21659.1,E2 -21659.1} C_VEL
LIN {X 0,Y 206.621,Z 606.458,A -85,B 0,C 180,E1 -21662.173,E2 -21662.173} C_VEL
LIN {X 0,Y 203.226,Z 610.879,A -85,B 0,C 180,E1 -21664.391,E2 -21664.391} C_VEL
LIN {X 0,Y 198.723,Z 616.515,A -85,B 0,C 180,E1 -21668.205,E2 -21668.205} C_VEL
